	(*****P14_BadBottleConyevor********)
	bBadBottleConveyorEnable						:BOOL;									//Zezwolenie na pracę transportera odrzuconych butelek
	nBadBottleConveyorVelocitySV					:UINT;									// Predkosc zadana transportera
	bBadBottleConveyorStart							:BOOL; 									// Zezwolenie na pracę transportera we/wy	

	(*******P14_TurnTable********)
	bExitTurnTableEnable							:BOOL;(**)								//Zezwolenie na pracę etykieciarki
	bExitTurnTableCmdStart 							:BOOL;
	bExitTurnTableGateRun							:BOOL;
	bExitConveyorEnable								:BOOL;(**)								//Zezwolenie na pracę 
	nExitConveyorVelocitySV							:UINT;
	bExitConveyorCmdStart 							:BOOL;
	bExitConveyorGateRun							:BOOL;

	
	(********P15_FormTransporters********)
	bFormTransportersEnable							:BOOL;			
	bFormTransportersDispencerCmdStart				:BOOL; 									// Start transporterów formatek w cyklu
	bFormTransportersBeforeROPPCmdStart				:BOOL;
	bFormTransportersScrewerCmdStart				:BOOL; 									// Start transporterów formatek w cyklu
	bFormTransportersScrewerStop					:BOOL; 									// Start transporterów formatek w cyklu
	bFormTransportersBeforeROPPStop					:BOOL;
	bFormTransportersDispencerSlowSpeedPulse		:BOOL;									// Wolna prędkość transportera
	bFormTransportersDispencerSlowSpeed				:BOOL;									// Wolna prędkość transportera
	bFormTransportersDispencerResetSpeed			:BOOL;									// Reset prędkości transportra
	ulFormTransportersScrewerSlowNumber				:ULINT;									// Nr RFID ostatniej formatki bez korka
	bFormTransportersAfterCapSorterCmdStart			:BOOL;									// Start transportera przez zakręcarka								// Aktywacja
	bFormTransportersBeforeScrewerCmdStart			:BOOL;									// Start transportera przez zakręcarka								// Aktywacja
	bFormTransporterSlowerCmdStart					:BOOL;									// Start transportera spowalniacza fomatek
	bFormTransportersAfterScrewerCmdStart			:BOOL;									// Start transportera przez zakręcarka								// Aktywacja
	ulSingleRealeseIfNoCapFromScrewersNumber		:ULINT;									// Nr RFID ostatniej formatki bez korka
	bSingleRealeseIfNoCapFromScrewersPulse			:BOOL;
	iSingleRealeseIfNoCapFromScrewersPulse			:INT;
				
	//Opcja z falownikiem
	nFormTransportersDispencerVelocitySV			:UDINT;		// Prędkość transportera otwartych butelek
	nFormTransportersScrewerVelocitySV				:UDINT;		// Prędkość transportera zamkniętych butelek
	nFormTransportersAfterCapSorterVelocitySV		:UDINT;		// Prędkość transportera przed zakręcarkami
	nFormTransportersBeforeScrewerVelocitySV		:UDINT;		// Prędkość transportera przed zakręcarkami
	nFormTransportersSlowerVelocitySV				:UDINT;		// Prędkość spowalniacza
	nFormTransportersAfterScrewerVelocitySV			:UDINT;		// Prędkość transportera przed zakręcarkami
	nFormTransportersROPPVelocitySV					:UDINT;		// Prędkość spowalniacza

	(******P16_LabelMachine********)
	bLabelMachineEnable								:BOOL;(**)								//Zezwolenie na pracę etykieciarki
	bLabelMachineCmdStart							:BOOL;		

	(*****P17_CircularInkJet********)
	bCircularInkjetEnable 							:BOOL;									// Zezwolenie na pracę Inkjet'u obwodowego	
	iCircularInkjetSpeed 							:INT;									// Prędkość rolek
	iCircularInkjetDelay							:INT;									// Opóźnienie docisku rolek
	iCircularInkjetHold								:INT;		
	
	bDragingFormsNotDone							:BOOL;				//Zmienna pomocnicza od przeciagania

	(**P20_ExhaustFan**)
	bExhaustFanEnable								:BOOL;
	bExhaustFanCmdStart								:BOOL;
	udiExhaustFanVelocitySV							:UDINT;
	


END_VAR

VAR_GLOBAL PERSISTENT
	(*****Zmienne presistent****)
	
	(***MAIN***)
	eRFID											:ARRAY [1..100] OF S_PackageState;		// STRUKTURA RFID
	AbRFIDFormOrder									:ARRAY [0..100] OF ULINT;				// Globalny rejestr kolejności formatek

	// Auton
	iDispencerRepair1								:INT;
	itonAfterDispencersRepair						:INT;
	itonAfterDispencersRepair1B						:INT;
	itonAfterDispencersRepair2						:INT;	
	itonAfterDispencersRepair3						:INT;	
	itonAfterDispencersRepair4						:INT;	
	itonRobotBottleTransferedToLabelerRepair		:INT;
	itonRobotBottleTransferedToLabeler2Repair		:INT;
	
	(***P00_Counters***)
	nGlobalCounterTemp								:UDINT;									//Tymczasowa zmienna do zapisywania licznika globalnego do pliku raz na jakiś czas
	
	(*Do diagnostyki*)
	iCounterDispencer34DosingAborted				:INT;
	iRepairFormBeforeDispenscerCounter				:INT;
	iRepairFormBeforeDispenscer2PhaseCounter		:INT;
	iRepairAfterDispencerCounter					:INT;
	iRepairBeforeDispencer12Counter					:INT;
	iRepairBeforeDispencer12Counter2				:INT;	
	iWeightRepair1Counter							:INT;
	iWeightRepair2Counter							:INT;
	iRepairFourthFormBeforeDispencerCounter			:INT;
	iRepairBeforeDispencer34Counter					:INT;
	
	iRepairLidFeeder1Counter						:INT;
	iRepairLidFeeder2Counter						:INT;
	iRepairLidFeeder3Counter						:INT;
	iRepairLidFeeder4Counter						:INT;
	
	iUnderScrewerPackageState222nCardNumberChangeCounter		: INT;
	iUnderScrewerPackageState333nCardNumberChangeCounter		: INT;
	iUnderScrewerPackageState111nCardNumberChangeCounter		: INT;
	
	iDispencerPackageState4nCardNumberChangeCounter	:INT;		
	iDispencerPackageState3nCardNumberChangeCounter	:INT;	
	iDispencerPackageState2nCardNumberChangeCounter	:INT;	
	iDispencerPackageState1nCardNumberChangeCounter	:INT;	
	
	iRobotPackageState2nCardNumberChangeCounter		:INT;	
	iRobotPackageState1nCardNumberChangeCounter		:INT;	
	
	iRobotRepairPackageForm1Counter					:INT;
	iRobotRepairPackageForm2Counter					:INT;	
	
	iScrewerFormStuck								:INT;
	iScrewerFormStuck2								:INT;
	iScrewerFormStuck3								:INT;

	(***MAIN***)
	//aSetIDBottle
	nID												:UDINT;									// Identycikacja butelek
		
	(*****P02_Dispencers****)
	bTank1LevelSensorCalibrated						:BOOL;									//Czujnik poziomu nr 1 skalibrowany	
	
	(*****P13_BottleTransfer********)
	nBottleTransferLubricationCounter				:DINT;									//Licznik po którym wyświetla się ostrzeżenie o smarowaniu robota
	
	
END_VAR

// ---- GVLs/gvlChecks.TcGVL
(*
Nazwa:			GVL_Checks
Opis:			Zmienne do sprawdzania błędów
Wersja:			v0.1
Data:			2018-10-10
Autor:			DP
Urzadzenia:		
Konfiguracja:	
Info:
(*d*) - obslużone
*)

{attribute 'qualified_only'}
VAR_GLOBAL PERSISTENT
	dCheckBounds		: DINT;	(*Licznik przekroczen zakresu indexow, np. tablic*)
	dCheckDivDInt		: DINT;	(*Licznik prob dzielenia Dint przez 0*)
	dCheckDivLInt		: DINT; (*Licznik prob dzielenia LInt przez 0*)
	dCheckDivLReal		: DINT; (*Licznik prob dzielenia LREAL przez 0*)
	dCheckDivReal		: DINT; (*Licznik prob dzielenia REAL przez 0*)
	dCheckRangeSigned	: DINT;	(*Licznik przekroczen  liczby znakowej*)
	dCheckRangeUnsigned	: DINT; (*Licznik przekroczen  liczby bezznakowej*)
END_VAR

// ---- GVLs/gvlCommunication.TcGVL
VAR_GLOBAL
	
		(*****P01_BottleSorter********)	
		stBottleSorterWrite			AT %MB0		: ST_Communication;		//Wysyłane zmienne do BottleSorter	
		//stBottleSorterWrite		AT %Q*		: ST_Communication;		//Wysyłane zmienne do BottleSorter
		stBottleSorterRead			AT %I*		: ST_Communication;		//Odczytane zmienne z BottleSorter
		
		//Zapis ADS
		//nic nie potrzeba, sprawdzanie czy jest butelka 
		//jest przed dozownikami
		
		//Odczyt ADS
		//nic nie potrzeba, sprawdzanie czy jest butelka 
		//jest przed dozownikami	
		bBottleSorterDoor1Open						: BOOL;				// Drzwi 1 otwarte
		bBottleSorterDoor2Open						: BOOL;				// Drzwi 2 otwarte	
		bBottleSorterSystemDiagError				: BOOL;				// Bład systemu BottleSorter

		(*****P04_CapSorter********)	
		stCapSorterWrite			AT %MB2000	: ST_Communication;	//Wysyłane zmienne do CapSorter	
		//stCapSorterWrite			AT %Q*		: ST_Communication;		//Wysyłane zmienne do CapSorter	
		stCapSorterRead				AT %I*		: ST_Communication;		//Odczytane zmienne z CapSorter
		
		//Zapis ADS		
		bCapSorterRobotPlace					: BOOL;				// Nałóż nasadki	
		bCapSorterRobotBottleAndNoCap1			: BOOL;				// Jest butelka bez nasadki w formatce 1
		bCapSorterRobotBottleAndNoCap2			: BOOL;				// Jest butelka bez nasadki	w formatce 2
		bCapSorterRobotBottleAndNoCap3			: BOOL;				// Jest butelka bez nasadki w formatce 3
		bCapSorterRobotBottleAndNoCap4			: BOOL;				// Jest butelka bez nasadki w formatce 4
		bCapSorterRobotPreparePlace				: BOOL;				// Przygotuj nasadki 			
		bCapSorterBeforeRobotBottleAndNoCap1	: BOOL;				// Jest butelka bez nasadki w formatce 1 przed robotem
		bCapSorterBeforeRobotBottleAndNoCap2	: BOOL;				// Jest butelka bez nasadki	w formatce 2 przed robotem
		bCapSorterBeforeRobotBottleAndNoCap3	: BOOL;				// Jest butelka bez nasadki w formatce 3 przed robotem
		bCapSorterBeforeRobotBottleAndNoCap4	: BOOL;				// Jest butelka bez nasadki w formatce 4 przed robotem
		
		//Odczyt ADS
		bCapSorterRobotPlaceDone				: BOOL;				// Wykonano, formatki mogą odjechać			
		bCapSorterRobotForm1CapPutted			: BOOL;				// Nasadka nałożona
		bCapSorterRobotForm2CapPutted			: BOOL;				// Nasadka nałożona
		bCapSorterRobotForm3CapPutted			: BOOL;				// Nasadka nałożona
		bCapSorterRobotForm4CapPutted			: BOOL;				// Nasadka nałożona
		
		bCapSorterDoor1Open						: BOOL;				// Drzwi 1 otwarte
		bCapSorterDoor2Open						: BOOL;				// Drzwi 2 otwarte		
		bCapSorterDoor3Open						: BOOL;				// Drzwi 3 otwarte	
		bCapSorterDoor4Open						: BOOL;				// Drzwi 4 otwarte		
		
		bCapSorterEmergencyStopButton1Pressed	: BOOL;				// Drzwi 1 otwarte
		bCapSorterEmergencyStopButton2Pressed	: BOOL;				// Drzwi 2 otwarte		
		bCapSorterEmergencyStopButton3Pressed	: BOOL;				// Drzwi 3 otwarte	
		
		bCapSorterRobotPlaceAck					: BOOL;				// Potwierdzenie rozpoczęcia cyklu		
	
END_VAR

// ---- GVLs/GVL_CP.TcGVL

VAR_GLOBAL
	

	//MAIN/PACKML
	eCapPusherPackageState					:ARRAY [1..17] OF S_PackageState;		// [1..6] 

	(******P00_Alarms******)
	CapPusherGateError						:S_Error; 								// Szlaban
	CapPusherFeederError					:S_Error; 								// Podajnik
	CapPusherError							:S_Error;								// Wbijak

	(******P07_CapPusher********)	  

	//Szlaban
	bCapPusherGateRun						:BOOL;		

	//Podajnik
	bCapPusherFeederDoHoming				:BOOL;									// Wykonanie bazowania stacji podajnika 
	iCapPusherFeederTimeDelayOn				:INT; 										
	iCapPusherFeederTimeDelayOff			:INT; 
	iCapPusherFeederTimeToEmptySleeveError	:INT:=120;									// Czas do alarmu pustego rękawa 
	iCapPusherFeederCheckCountNOK			:INT;									// Zliczanie butelek bez nasadek

	//Zakrecanie
	bCapPusherDoHoming						:BOOL;									// Wykonanie bazowania stacji 
	bCapPusherEnable						:BOOL:=TRUE; 	
	iCapPusherTime							:INT; 	
	iCapPusherTime2							:INT;	

END_VAR

(*
VAR_GLOBAL PERSISTENT
	iRepairROPP1Counter						:INT;
	iRepairROPP2Counter						:INT;
	iRepairROPP3Counter						:INT;
	iRepairROPP4Counter						:INT;
END_VAR	*)

// ---- GVLs/GVL_IO.TcGVL
(*
Nazwa:			GVL_IO
Opis:			Zmienne I/O nie wykorzystywane w blokach stacji
Wersja:			v0.1
Data:			2018-10-10
Autor:			DP
Urzadzenia:		
Konfiguracja:	
Info:
(*d*) - obslużone
*)


VAR_GLOBAL

(*Safety ##############################*)
	//Przesylane, odbierane z/do SafetyPLC
	IbEmergencyStopButton 	AT %I*		: BOOL; 		//Jeśli FALSE - Estop wysyołany przez przyciski
	IbEmergencyStop 		AT %I* 		: BOOL; 		//Jeśli TRUE - maszyna w stanie bezpiecznym, FALSE - EStop
	IbBottleFeederSafety	AT %I*		: BOOL;			// Status Safety z podajnika butelek
	IbSafetyResetIn			AT %I*		: BOOL;			// Przycisk Reset
	QbSafetyResetCapSorterIn AT %Q*		: BOOL;			// Przycisk Reset
	QbSafetyResetBottleSorterIn AT %Q*	: BOOL;			// Przycisk Reset
	QbSafetyResetDelay 		AT %Q*		: BOOL;			// Zezwolenie na pierwsze zresetowanie
	
	
	IbCommunicationErrorUF50	AT %I* 	:BOOL;			//Do alarmu komunikacji z safety
	IbCommunicationErrorUP50B	AT %I* 	:BOOL;			//Do alarmu komunikacji z safety
	
	IbBottleSorterDisable		AT %I* 	:BOOL:=TRUE;			//Sygnał z kluczyka blokady safety
	IbCapSorterDisable			AT %I* 	:BOOL:=TRUE;			//Sygnał z kluczyka blokady safety

	
(*Wejscia ogólne #####################*)

	IbPowerSupplyOK 				AT %I*		:BOOL;		//Napięcie zasilania OK
	IbDCSupply1OK 					AT %I*		:BOOL;		//Zasilacz alarm	
	IbFuseFB1OK						AT %I*		:BOOL;		//Bezpiecznik FB1 przepalony
	IbDCSupply2OK					AT %I*		:BOOL;		//Zasilacz alarm	
	IbFuseFB2OK						AT %I*		:BOOL;		//Bezpiecznik FB2 przepalony
	IbDCSupply3OK					AT %I*		:BOOL;		//Zasilacz alarm	
	IbFuseDrivesOK					AT %I*		:BOOL;		//Bezpiecznik Servonapędów
	IbFuseFormTransporter1OK		AT %I*		:BOOL;		//Bezpiecznik silnikowe napędu transportera 1
	IbFuseFormTransporter2OK		AT %I*		:BOOL;		//Bezpiecznik silnikowe napędu transportera 2
	IbFuseFormTransporter3OK		AT %I*		:BOOL;		//Bezpiecznik silnikowe napędu transportera 3 (odrzuty)
	IbFuseFormTransporter4OK		AT %I*		:BOOL;		//Bezpiecznik silnikowe napędu transportera 4 (spowalniacz)
	IbFuseFormTransporter5OK		AT %I*		:BOOL;		//Bezpiecznik silnikowe napędu transportera 4 (33F1)
	IbFuseFormTransporter6OK		AT %I*		:BOOL;		//Bezpiecznik silnikowe napędu transportera 4 (34F1)
	IbBottleFeederTurntableOK		AT %I*		:BOOL;		//Zabezpieczenie silnikowe stolu obrtooergo
	IbDCSupply4OK					AT %I*		:BOOL;		//Zasilacz alarm			
	IbDCSupply5OK					AT %I*		:BOOL;		//Zasilacz alarm		
	IbFuseFB3OK						AT %I*		:BOOL;		//Bezpiecznik FB3 przepalony
	IbDC5VSupply1OK 				AT %I*		:BOOL;		//Zasilacz 5V alarm	

	
	IbLinearPowerSupplyOK			AT %I*		:BOOL;	
	IbStepperPowerSupplyOK			AT %I*		:BOOL;	
	IbFuseFanEXMotor				AT %I*		:BOOL;	
	IbStepperMotorsFuseOK			AT %I*		:BOOL;
	IbFuse10F9OK					AT %I*		:BOOL;
	IbFuse10F11OK					AT %I*		:BOOL;
	
	//IbFuseTankMixerEngineOK w Dispencers
	IbTanksDoorsOpen 				AT %I*		:BOOL;		//Otwarte drzwi pod zbiornikami
	IbLidSealingDoorsOpen			AT %I*		:BOOL;		//Otwarte drzwi przygrzewaczki
	IbGripperScrewerDoorsOpen		AT %I*		:BOOL;		//Otwarte drzwi przy zakrecarkach
	IbDispencersDoorsOpen 			AT %I*		:BOOL;		//Otwarte drzwi przy dozownikach
	IbBottleTransferDoorsOpen		AT %I*		:BOOL;		//Otwarte drzwi z boku dozowników

	IbEmergencyStopButton0Pressed	AT %I*		:BOOL;		//Przyciśnięty przycisk E-Stop0	Pulpit główny przod
	IbEmergencyStopButton1Pressed	AT %I*		:BOOL;		//Przyciśnięty przycisk E-Stop1 przy transporterze odrzuconych opakowań
	IbEmergencyStopButton2Pressed	AT %I*		:BOOL;		//Przyciśnięty przycisk E-Stop2 przy drzwiach robota
	IbEmergencyStopButton3Pressed	AT %I*		:BOOL;		//Przyciśnięty przycisk E-Stop3 przy zakręcarkach
	IbEmergencyStopButton4Pressed	AT %I*		:BOOL;		//Przyciśnięty przycisk E-Stop4	Pulpit tylny

	// podajnik butelek
	
	IbBottleFeederSafetyDoor1Open	AT %I*		:BOOL;		// Czujnik otwarcia drzwi dostępowych 
	IbBottleFeederSafetyDoor2Open	AT %I*		:BOOL;		// Czujnik otwarcia drzwi dostępowych drugie
	IbBottleFeederSafetyDoor3Open	AT %I*		:BOOL;		// Czujnik otwarcia drzwi dostępowych drugie
	
	
	//Vasyl 28.05
	IbPucksInserterRollerFuse		 AT %I*      :BOOL;		// Zabezpieczenie 71F4 Rolka obracająca
	IbPucksInserterPushTableFuse	 AT %I*      :BOOL;		// Zabezpieczenie 71F3 Stół podający
	IbEmergencyStopButtonPushtable1  AT %I*		:BOOL;
	IbEmergencyStopButtonPushtable2  AT %I*		:BOOL;
	
	
	IbCycleStartButton				AT %I*		:BOOL;		//Przycisk Startu cyklu
	//IbSafetyResetIn				AT %I*		:BOOL;		//Reset
	IbCycleStopButton				AT %I*		:BOOL;		//Przycisk Stopu cyklu
	//IbTank1LevelLow w Dispencers
	//IbTank2LevelLow w Dispencers
	IbCompressedAirOK 				AT %I*		:BOOL;		//Zasilanie powietrzem sprężonym OK	
	
(* I/O robot*)
	//Alarm zasilacz DC1 w BottleTransfer
	//Bezpiecznieki OK w BottleTransfer

	IbFuseCircularInkjetOK			AT %I*		:BOOL;		//Zabezpieczenie silnikowe InkJet obwodowy	
	
	QbResetFuseFB1					AT %Q*		:BOOL;	
	QbResetFuseFB2					AT %Q*		:BOOL;
	QbResetFuseFB3					AT %Q*		:BOOL;	

(* Diagnostyka modułów*)
	IbPowerSuppyTerminal1UpUndervoltage	AT %I*		:BOOL;	{warning 'dodać alarm'}// Brak napięcia zasilania na module ST1 w szafie głównej
	IbPowerSuppyTerminal1UsUndervoltage	AT %I*		:BOOL;	
	IbPowerSuppyTerminal2UpUndervoltage	AT %I*		:BOOL;	// Brak napięcia zasilania na module ST1 w szafie robota
	IbPowerSuppyTerminal2UsUndervoltage	AT %I*		:BOOL;	// Brak napięcia E-Bus na module ST1 w szafie robota
	
	QbDispencersDoorsClose				AT %Q*		:BOOL;		// Rozkaz zamkniecia 
	QbGripperScrewerClose				AT %Q* 		:BOOL;		// Rozkaz zamkniecia 
	QbBottleTransferDoorsClose			AT %Q*		:BOOL; 		// Rozkaz zamkniecia 
	QbTanksDoorsClose 					AT %Q*		:BOOL;		// Rozkaz zamkniecia
	QbLidSealingDoorsClose				AT %Q*		:BOOL;		// Rozkaz zamkniecia
	
	(*Wybdmuch nakretek*)
	QbBlowAfterGripperScrewer						: BOOL; 
	QbBlowBeforeGripperScrewer						: BOOL; 
	IbBlowBeforeGripperScrewerSensor				: BOOL;
	QbGateBeforeGripperScrewer						: BOOL;	
	IbGateBeforeGripperScrewerSensor				AT %I*		:BOOL;	

	//Dodatkowy szlaban przed zakrecarka
	QbGripperScrewerStoperActuator			:BOOL;	//Stoper
	QbGripperScrewerStoper2Actuator			:BOOL;	//Stoper krótki
	QbGripperScrewerGateBeforeActuator		:BOOL;	//Szlaban
	//Koniec Dodatkowy szlaban przed zakrecarka

	//Dodatkowy szlaban za robotem
	QbBottleTransferAfterDragActuator		:BOOL;	//Stoper
	QbBottleTransferAfterDragStoperActuator	:BOOL;	//Stoper krótki
	QbBottleTransferAfterDragGateActuator	:BOOL;	//Szlaban
	//Koniec Dodatkowy szlaban za robotem


	
	//Dodatkowy popychacz za zakręcarką
	QbGripperScrewerAcceleratorActuator			:BOOL;
	
	(*I/O TurnTable*)
	IbTurnTableSafety						AT %I*		:BOOL;		//Przyciśnięty przycisk E-Stop0	Pulpit główny
	IbTurnTableMotorOK						AT %I*		:BOOL;		//Zabezpieczenie silnikowe stolu obrtooergo 
	IbTurnTableEmergencyStopButtonPressed	AT %I*		:BOOL;		//Przyciśnięty przycisk E-Stop0	Pulpit główny
	IbTurnTableCycleStartButton				AT %I*		:BOOL;		//Przycisk Startu cyklu
	IbTurnTableCycleStopButton				AT %I*		:BOOL;		//Przycisk Stopu cyklu
	IbTurnTableFuseProtection				AT %I*		:BOOL;		//Zabezpieczenie stół obrotowy

	IbExitConveyorOK						AT %I*		:BOOL;		//Zabezpieczenie silnikowe stolu obrtooergo


	(*I/O PI*)
	IbPucksInserterDoorsOpen	{warning 'PI'}	AT %I*		:BOOL;		//Otwarte drzwi podajnika opakowań
	QbPickInserterDoorsClose	{warning 'PI'}	AT %Q*		:BOOL;		// Rozkaz zamkniecia 
	IbPucksInserterEmergencyStopButton0Pressed	AT %I*		:BOOL;		//Przyciśnięty przycisk E-Stop0	
	IbPucksInserterEmergencyStopButton1Pressed	AT %I*		:BOOL;		//Przyciśnięty przycisk E-Stop1	
	IbPucksInserterCycleStartButton				AT %I*		:BOOL;		//Przycisk Startu cyklu
	IbPucksInserterCycleStopButton				AT %I*		:BOOL;		//Przycisk Stopu cyklu

(* IO wybychowe**)
	
	IbExModeSwitchNormalMode		AT %I*		:BOOL;		// Wybór trybu pracy - tryb zwykły
	IbExModeSwitchExMode			AT %I*		: BOOL;		// Wybór trybu pracy - tryb pracy wybuchowej
	
	
(* Czujnik ciśnienia w układzie *)
	IbPressureInSystemSensor		AT %I*	:BOOL;
	

END_VAR

// ---- GVLs/GVL_ROPP.TcGVL

VAR_GLOBAL
	

	//MAIN/PACKML
	eBeforeROPPCapControlPackageState		:ARRAY [1..17] OF S_PackageState;		// [1..1] 
	eBeforeROPPPackageState					:ARRAY [1..17] OF S_PackageState;		// [1..6] 
	eBeforeROPP2PackageState				:ARRAY [1..17] OF S_PackageState;		// [1..6] 
	eUnderROPPPackageState 					:ARRAY [1..17] OF S_PackageState;		// [1..3] 
	eUnderROPPCorrectCapPackageState		:ARRAY [1..17] OF S_PackageState;		// [1..7] 

	(******P00_Alarms******)
	ROPPSlowerError							:S_Error; 								// Spowalniacz
	ROPPFeederError							:S_Error; 								// Spowalniacz
	ROPPDragError							:S_Error;								// 14 
	ROPPCappingError						:S_Error;								// 14 

	(******P07_ROPP********)	  

	//Spowalniacz
	bROPPSlowerEnable						:BOOL:=TRUE;			
	bROPPSlowerCmdStart						:BOOL:=TRUE;									// Start transportera spowalniacza fomatek
	nROPPSlowerVelocitySV					:UDINT:=2100;	

	//Podajnik
	bROPPFeederDoHoming						:BOOL;									// Wykonanie bazowania stacji podajnika 
	bROPPFeederEnable						:BOOL; 	
    lrROPPFeederHeightPosSV					:LREAL;									 	
	iROPPFeederTimeDelayOn					:INT; 										
	iROPPFeederTimeDelayOff					:INT; 
	iROPPFeederTimeToEmptySleeveError		:INT;									// Czas do alarmu pustego rękawa 
	iROPPFeederCheckCountNOK				:INT;									// Zliczanie butelek bez nasadek

	//Przeciąganie formatek 
	aROPPDragAxisRef						:AXIS_REF;								// Struktura osi napędu krokowego przeciągania	
	bROPPDragEnable							:BOOL;									// Zezwolenie na pracę przeciągania 
	bROPPDragDoHoming						:BOOL;									// Wykonanie bazowania przeciągania
	bROPPDragHeightSet						:BOOL;									// Wykonanie bazowania przeciągania
	bROPPDragPrepareRun						:BOOL;
	lrROPPDragVelocity						:LREAL:=100;							// Prędkośc przeciągania
	lrROPPDragAcceleration					:LREAL:=12;								// Przyspieszenie przeciągania
	lrROPPDragDeceleration					:LREAL:=15;								// Hamowanie przeciągania

	//Zakrecanie
	bROPPCappingRunEngine					:BOOL;									
	bROPPCappingDoHoming					:BOOL;									// Wykonanie bazowania stacji 
	bROPPCappingEnable						:BOOL; 	
    lrROPPCappingHeightPosSV				:LREAL;									 	
	lrROPPCappingVelocitySV					:UDINT;	
	iROPPCappingTime						:INT; 	
	iROPPCappingTime2						:INT;	
	iROPPCapping1Tool						:INT;									// Wybór narzędzia (1-5), opisy w tablicy AsGripperScrewerTool	

END_VAR

(*
VAR_GLOBAL PERSISTENT
	iRepairROPP1Counter						:INT;
	iRepairROPP2Counter						:INT;
	iRepairROPP3Counter						:INT;
	iRepairROPP4Counter						:INT;
END_VAR	*)

// ---- GVLs/GVL_RS.TcGVL

VAR_GLOBAL
	
	//MAIN/PACKML
	eRollerScrewerPackageState					:ARRAY [1..17] OF S_PackageState;		// [1..6] 

	(******P00_Alarms******)
	RollerScrewerGateError						:S_Error; 								
	RollerScrewerError							:S_Error;								
	RollerScrewerCatchError						:S_Error;								
                                                                                        
	(*****P11_RollerScrewer********)  
	//Szlaban
	bRollerScrewerGateRun						:BOOL;		
	//Zakrecanie
	bRollerScrewerDoHoming						:BOOL;									// Wykonanie bazowania stacji podajnika 
	//Ciśnienia - nie wiadomo czy będą
	lrRollerScrewerCatchPressure 				:LREAL;			
	lrRollerScrewerPressingRollsPressure		:LREAL;			
	lrRollerScrewerPressingTopPressure 			:LREAL;			
	//Zakręcarka rolkowa
	aRollerScrewerFrontAxisRef					: AXIS_REF;									// Struktura NC napędu zakręcarki rolkowej
	aRollerScrewerRearAxisRef					: AXIS_REF;									// Struktura NC napędu zakręcarki rolkowej
	bRollerScrewerEnable						: BOOL;			
	bRollerScrewerFindScrew						: BOOL; 		
	lrRollerScrewerFindingScrewDegree			: LREAL; 		
	lrRollerScrewerVelocity						: LREAL:=50; 
	iRollerScrewerTightTime						: INT:=100;  
	lrRollerScrewingTightTorque					: LREAL;  		
    lrRollerScrewerHeightPosSV					: LREAL:=72;	
	uiRollerScrewerTopActuatorTimeDelayOff		: UINT;  		
	//Chwytak zakręcarki rolkowej                               		
	lrRollerScrewerCatchHeightSV				: LREAL:=36; 
	bRollerScrewerCatchRun						: BOOL; 
	bRollerScrewerCatchDoHoming					: BOOL; 

	
END_VAR

(*
VAR_GLOBAL PERSISTENT
	iRepairROPP1Counter						:INT;
	iRepairROPP2Counter						:INT;
	iRepairROPP3Counter						:INT;
	iRepairROPP4Counter						:INT;
END_VAR	*)

// ---- GVLs/Iterators.TcGVL
VAR_GLOBAL
	i								: INT;
END_VAR

// ---- GVLs/UVFF/GVL_Recipe.TcGVL
(*
Nazwa:			GVL_Recipe
Opis:			Zmienne recepturowe tylko do wizualizacji
Wersja:			v0.2
Data:			2024-02-20
Autor:			MK
Urzadzenia:		
Konfiguracja:	
Info:
Zmiany:
- 20240220 [DP] Poprawki przed nowa wizką
*)
VAR_GLOBAL
	(*Legenda dla wizki :
		[H] - Hidden, prawdopodobnie nie potrzebne
		[I] - Info, informacja,
		[L] - Later, do zrobienia później, być może do przerobienia
		Uprawienia:
		brak opisu - operator
		[m] - Meechanik i powyżej
		[t] - Technolog i powyżej
		[s] - Serwis i powyżek
		[a] - Admin			
	*)	
	
	//Sorter nasadek, typ produktu	
	iCapSorterProductType										: INT		:= 2; 		//		Typ produktu: 0- kule/fliptopy, 1- pompki, 2- disctop, 3-airless, 4-decoration cap (wyłączone podcisnienie na załapywarce), 5- decoration cap with new gripper (wyłączone podcisnienie + nowy program do robota)
	uiCapSorterIndexShow										: UDINT		:= 5;		//		Index produktu	
	bPresenceBottleEnableShow									: BOOL;					//		Sprawdzanie butelki w formatce

//--------------------------------------CapSorterTransporter-----------------------------------------------------------------------------------------------------------------------------	
	// Sorter nasadek, transporter zasobnika
	bCapSorterTransporterEnableShow								: BOOL;					//		Aktywacja
	iCapSorterTransporterTankConveyorVelocityShow				: INT		:= 1200;	//		Prędkość 							| [%] (1.0-100.0)
	iCapSorterTransporterStartDelayTimeShow						: INT		:= 100;		//		Timer do załączania 				| [ms] (0.0-10_000.0)
	udiCapSorterTransporterTimeProductOnSensorBeforeBrushShow	: UDINT		:= 150;		//		Timer pracy							| [ms] (0.0-10_000.0)
	iCapSorterTransporterEmptyingConveyorSpeedShow				: INT		:= 25;		// 		Prędkość, opróżnianie 				| [%] (1.0-100.0)
	iCapSorterTransporterVolumeOfCapsShow						: INT		:= 330;		//		Odłegłość do zamknięć, ostrzeżenie 	| [mm] (0.0-10_000.0)

//---------------------------------------CapSorterWheel----------------------------------------------------------------------------------------------------------------------------	
	// Sorter nasadek, stól
	bCapSorterWheelEnableShow									: BOOL;					//		Aktywacja
	lrCapSorterWheelMoveAccelerationEmptyTableShow				: LREAL		:= 5000;	//		Dynamika rozpędzania - pusty 		| [obr/min²], (1.0-100_000.0) 
	lrCapSorterWheelMoveDecelerationEmptyTableShow				: LREAL		:= 5000;    //		Dynamika spowalniania - pusty 		| [obr/min²] (1.0-100_000.0) 
	lrCapSorterWheelMoveSpeedEmptyTableShow						: LREAL		:= 334;     //		Prędkość - pusty 					| [obr/min] (1.0-10_000.0)                
	lrCapSorterWheelMoveAngleEmptyTableShow						: LREAL		:= 20;      //		Kąt - pusty 						| [obr/min] (0.0-360.0)                        
	lrCapSorterWheelJerkAngleEmptyTableShow						: LREAL		:= 15000;   //		Zryw - pusty 						| [obr/min³] (1.0-1_000_000)                  
	iCapSorterWheelWaitingAfterRotationEmptyTableShow			: INT		:= 100;     //		Czas stabilizacji - pusty 			| [ms] (0.0-1_000)                 
	
	lrCapSorterWheelMoveAccelerationFullTableShow				: LREAL		:= 5000;	//		Dynamika rozpędzania - pełny 		| [obr/min²], (1.0-100_000.0) 
	lrCapSorterWheelMoveDecelerationFullTableShow				: LREAL		:= 5000;    //		Dynamika spowalniania - pełny 		| [obr/min²] (1.0-100_000.0) 
	lrCapSorterWheelMoveSpeedFullTableShow						: LREAL		:= 334;     //		Prędkość - pełny 					| [obr/min] (1.0-10_000.0)                
	lrCapSorterWheelMoveAngleFullyTableShow						: LREAL		:= 6;       //		Kąt - pełny 						| [obr/min] (0.0-360.0)                        
	lrCapSorterWheelJerkAngleFullTableShow						: LREAL		:= 15000;   //		Zryw - pełny 						| [obr/min³] (1.0-1_000_000)                  
	iCapSorterWheelWaitingAfterRotationFullTableShow			: INT		:= 30;      //		Czas stabilizacji - pełny 			| [ms] (0.0-1_000)                 
	
	lrCapSorterWheelMoveAccelerationHalfFullTableShow			: LREAL		:= 5000;	//		Dynamika rozpędzania - półpełny 	| [obr/min²], (1.0-100_000.0) 
	lrCapSorterWheelMoveDecelerationHalfFullTableShow			: LREAL		:= 5000;    //		Dynamika spowalniania - półpełny 	| [obr/min²] (1.0-100_000.0) 
	lrCapSorterWheelMoveSpeedHalfFullTableShow					: LREAL		:= 334;     //		Prędkość - półpełny 				| [obr/min] (1.0-10_000.0)                
	lrCapSorterWheelMoveAngleHalfFullyTableShow					: LREAL		:= 12;      //		Kąt - półpełny						| [obr/min] (0.0-360.0)                        
	lrCapSorterWheelJerkAngleHalfFullTableShow					: LREAL		:= 15000;   //		Zryw - półpełny 					| [obr/min³] (1.0-1_000_000)                  
	iCapSorterWheelWaitingAfterRotationHalfFullTableShow		: INT		:= 50;      //		Czas stabilizacji - półpełny 		| [ms] (0.0-1_000)               
	
//-------------------------------------CapSorterCamera------------------------------------------------------------------------------------------------------------------------------	                                                    	
	// Sorter nasadek, system wizyjny
	
    bCapSorterCameraEnableShow									: BOOL; 				//	[H]	Aktywacja                            	
	
//-----------------------------------------CapSorterRobot--------------------------------------------------------------------------------------------------------------------------	
	// Sorter nasadek, robot
	bCapSorterRobotEnableShow									: BOOL;					//		Aktywacja
                                                                                                                           	
	lrCapSorterRobotPlace1PositionXShow							: LREAL;				//		Offset odkładania 1, X 			| [mm]	((-100.0)-100.0)       
	lrCapSorterRobotPlace1PositionYShow							: lreal;    			//		Offset odkładania 1, Y 			| [mm]	((-100.0)-100.0)       
	lrCapSorterRobotPlace1PositionZShow							: lreal;    			//		Offset odkładania 1, Z 			| [mm]	((-100.0)-100.0)       
	lrCapSorterRobotPlace1PositionCShow							: lreal;    			//		Offset odkładania 1, C 			| [° ]	((-360.0)-360.0)                 
	iCapSorterRobotPickElevationShow							: INT;					//		Punkt nad poz. Pick				| [mm]	(30-1000)
	iCapSorterRobotPickTimeShow									: INT;					//		Czas przyssania					| [ms]	(0-10_000)
	iCapSorterRobotVacuumActivationShow							: INT;					//		Czas przed przyssaniem			| [ms]	(0-1000)
	iCapSorterRobotVacuumOffShow								: INT;					//		Czas przed oddmuchem			| [ms]	(0-1000)
	iCapSorterRobotPlaceTimeShow								: INT;					//		Czas oddmuchu					| [ms]	(0-1000)
	iCapSorterRobotTCP_PlaceOffsetShow							: INT;					//		Wysokość od TCP do p. odłożenia	| [mm]	(0-1000)									
	iCapSorterRobotAccelerationDecelerationShow					: INT;					//		Dynamika rozpędzania/hamowania	| [%]	(20-100)
	iCapSorterRobotGripperWatchdogShow							: INT;					//		Czas sprawdzania silownika		| [ms]	(0-1000)
	iCapSorterRobotParalaxCorrectionShow						: INT;					//		Korekta paralaxy				| [mm]	(0-100)
	
	iCapSorterRobotNumberToolShow								: INT;					//		Numer narzędzia					| 		(0-10)
	iCapSorterRobotPickPositionZShow							: INT;					//		Wysokość pobierania 			| [mm]	(0-200)
	iCapSorterRobotTCP_Lenght									: INT;					//		Długość chwytaka				| [mm]	(10-100)
	iCapSorterRobotProductDiametr								: INT;					//		Średnica nasadki				| [mm] 	(10-100)
	
//----------------------------------------CapSorterIntermediateTransporter---------------------------------------------------------------------------------------------------------------------------
	// Sorter nasadek, transporter zasypowy
	bCapSorterIntermediateTransporterEnableShow					: BOOL;					//		Aktywacja
	iCapSorterIntermediateTransporterAutoSpeedShow				: INT		:= 20;		//		Prędkość 					| [%] (1.0-100.0)
	iCapSorterIntermediateTransporterManualSpeedShow			: INT		:= 30;		//		Prędkość, manual 			| [%] (1.0-100.0)
	iCapSorterIntermediateTransporterEmptyingSpeedShow			: INT		:= 50;		//		Prędkość, opróżnianie 		| [%] (1.0-100.0)
	iCapSorterIntermediateTransporterDelayCountTimeShow			: INT		:= 100;		//		Timer pracy					| [ms]	(0.0-100_000.0)
	iCapSorterIntermediateTransporterReverseTimeShow			: INT		:= 4000;	//		Timer odwróconej pracy 		| [ms] (0.0-10_000.0)
	udiCapSorterIntermediateTransporterTimeProductOnSensorShow	: UDINT		:= 1800;	//		Czas produktu na czujniku 	| [ms] (0.0-10_000.0)	
	lrCapSorterIntermediateTransporterWheelAngleShow			: LREAL		:= 6;		//		Kąt zasypu 					| [°] (1.0-360.0)
	lrCapSorterIntermediateTransporterItemsSetValueShow			: LREAL	;				// 		Ilość detali na kołe		| []
	
//----------------------------------------CapSorterIntermediateBrush---------------------------------------------------------------------------------------------------------------------------
	//Sorter nasadek, szczotka transportera
	bCapSorterIntermediateBrushEnableShow						: BOOL;					//		Aktywacja
	iCapSorterIntermediateBrushAutoSpeedShow					: INT		:= 30;		//		Prędkość  					| [%] (0.0-100.0)
	iCapSorterIntermediateBrushManualSpeedShow					: INT		:= 30;		//		Prędkość, manual 			| [%] (0.0-100.0)
	iCapSorterIntermediateBrushEmptyingSpeedShow				: INT		:= 30;		//		Prędkość, opróżnianie 		| [%] (0.0-100.0)
	lrCapSorterIntermediateBrushPositionHeightSVShow			: LREAL		:= 45;		//		Wysokość 					| [mm] (0.0-10_000.0)

//----------------------------------------CapSorterBrush1OnWheel---------------------------------------------------------------------------------------------------------------------------
	// Sorter nasadek, szczotka stolu 1
	bCapSorterBrush1OnWheelEnableShow							: BOOL;					//		Aktywacja
	iCapSorterBrush1OnWheelAutoSpeedShow						: INT		:= 30;		//		Prędkość 					| [%] (0.0-100.0)
	iCapSorterBrush1OnWheelManualSpeedShow						: INT		:= 30;		//		Prędkość, manual 			| [%] (0.0-100.0)
	iCapSorterBrush1OnWheelEmptyingSpeedShow					: INT		:= 30;		//		Prędkość, opróżnianie 		| [%] (0.0-100.0)
	lrCapSorterBrush1OnWheelPositionHeightSVShow				: LREAL		:= 45;		//		Wysokość 					| [mm] (0.0-10_000.0)
	
//----------------------------------------CapSorterBrush2OnWheel----------------------------------------------------------------------------------
	// Sorter nasadek, szczotka stolu 2
	bCapSorterBrush2OnWheelEnableShow							: BOOL;					//		Aktywacja
	iCapSorterBrush2OnWheelAutoSpeedShow						: INT		:= 30;		//		Prędkość 					| [%] (0.0-100.0)
	iCapSorterBrush2OnWheelManualSpeedShow						: INT		:= 30;		//		Prędkość, manual 			| [%] (0.0-100.0)
	iCapSorterBrush2OnWheelEmptyingSpeedShow					: INT		:= 30;		//		Prędkość, opróżnianie 		| [%] (0.0-100.0)
	lrCapSorterBrush2OnWheelPositionHeightSVShow				: LREAL		:= 45;		//		Wysokość 					| [mm] (0.0-10_000.0)

//------------------------------------------CapFeeder-------------------------------------------------------------------------------------------------------------------------	
	// Sorter nasadek, 
	bCapSorterFeederEnableShow									: BOOL;					//		Aktywacjaa
	bCapSorterFeederEnableTubeError								: BOOL;					// 		Aktywacja błedu słomki
	lrCapSorterFeederMover1InputPositionShow					: LREAL;				//		Pozycja wkładania, wózek 1 	| [mm] (?-?)
	lrCapSorterFeederMover2InputPositionShow					: LREAL;				//		Pozycja wkładania, wózek 2 	| [mm] (?-?)
	lrCapSorterFeederMover1OutputPositionShow					: LREAL;				//		Pozycja wyjmowania, wózek 1 | [mm] (?-?)
	lrCapSorterFeederMover2OutputPositionShow					: LREAL;				//		Pozycja wyjmowania, wózek 2 | [mm] (?-?)
	lrCapSorterFeederSlotDistanceShow							: LREAL;				//		Offset wkładania			| [mm] (?-?)			Old-(Odstęp między pozycjami kładzenia)
	lrCapSorterFeederMoverSpeedShow								: LREAL;				//		Prędkość				 	| [%] (0.0-100.0)
	lrCapSorterFeederMoverAccelerationShow						: LREAL;				//		Przyspieszenie 				| [mm/s²] 
	lrCapSorterFeederMoveJerkShow								: LREAL;				//		Zryw						| [mm/s³]

//-------------------------------------------------------------------------------------------------------------------------------------------------------------------	
	//CapPreScrewer		
	bCapSorterPreScrewerEnableShow								: BOOL;					// 		Aktywacja
	bCapSorterPreScrewerPicker1EnableShow						: BOOL;					// 		Aktywacja	
	bCapSorterPreScrewerPicker2EnableShow						: BOOL;					// 		Aktywacja
	bCapSorterPreScrewerPicker3EnableShow						: BOOL;					// 		Aktywacja	
	bCapSorterPreScrewerPicker4EnableShow						: BOOL;					// 		Aktywacja
	//Oś Z
	lrCapSorterPreScrewerPickZPositionShow						: LREAL;				//		Wysokość pobierania						| [mm]	
	lrCapSorterPreScrewerCatcherReleseShow						: LREAL;				//		nie używamy Wysokość otwierania chwytaka nakrętek	| [mm]		
	lrCapSorterPreScrewerCapCatcherZPositionShow				: LREAL;				//		Wysokość zamykania nakrętkek			| [mm]
	lrCapSorterPreScrewerTopZPositionShow						: LREAL;				//		Pozycja górna ośi Z						| [mm] 	
	lrCapSorterPreScrewerCartesianCatchZPositionShow			: LREAL; 				//      Wait Position
	lrCapSorterPreScrewerStrawCatcherZPositionShow				: LREAL;				//		Wysokość otwierania łapaczy słomek		| [mm]	
	LrCapSorterPreScrewerCheckStrawCatcherActuatorZPosition		: LREAL;				//		Wysokość sparawdzania cofania łapaczy słomek	| [mm]	
	lrCapSorterPreScrewerScrewerStartZPositionShow				: LREAL;				//		Wysokość początku zakręcania			| [mm]	
	lrCapSorterPreScrewerGripperOpenPositionShow				: LREAL;				//		Pozycja otwierania chwytaka butelek 	| [mm]
	lrCapSorterPreScrewerPlaceZPositionShow						: LREAL;				//		Wysokość odkładania - koniec załapywania gwintu	| [mm] 

	lrCapSorterPreScrewerThreadPitchShow						: LREAL;				//		Skok gwintu 		| [mm]	
	lrCapSorterPreScrewerMultipleStartThreadShow				: LREAL;				//		Krotność gwintu
	lrCapSorterPreScrewerNumberOfThreadTurnsShow				: LREAL;				//		Ilość obrotów
  	
	//Wspólne ruchi	
	lrCapSorterPreScrewerBendingDistanceShow					: LREAL;				//		Odległość zaokrąglania ruchów 			| [mm]		
	lrCapSorterPreScrewerStrawInsertDistance					: LREAL;				//		Odległość wspólnego ruchu, prowadzenie słomki	| [mm]		
	//Oś x
	lrCapSorterPreScrewerPickXMover1PositionShow				: LREAL;				//		Pozycja osi poziomej do pobierania, wozek 1	| [mm]
	lrCapSorterPreScrewerPickXMover2PositionShow				: LREAL;				//		Pozycja osi poziomej do pobierania, wozek 2	| [mm]
	lrCapSorterPreScrewerPlaceXPositionShow						: LREAL;				//		Pozycja osi poziomej do odkładania			| [mm]
	//Oś zakręcania
	lrCapSorterPreScrewerScrewFindingShow						: LREAL;				//		Kąt szukania gwintu							| [°]
	lrCapSorterPreScrewerScrewDistanceShow						: LREAL;				//		Kąt zakręcania								| [°]
	//Prédkośći                                                                                                                         	
	lrCapSorterPreScrewerPickerSpeedShow						: LREAL;				//		Prędkość									| [%]   
	lrCapSorterPreScrewerPickerSpeedWhenScrewerShow				: LREAL;				//		Prędkość osi Z przy zakręcaniu				| [%]   
	lrCapSorterPreScrewerPickerAccelerationShow					: LREAL;				//		Przyspieszenie								| [mm/s²] 		
	lrCapSorterPreScrewerPickerJerkShow							: LREAL;				//		Zryw										| [mm/s³]
                                                                                                                                        	
	lrCapSorterPreScrewerCatcherSpeedShow						: LREAL;				//		Prędkość									| [mm/s] 
	lrCapSorterPreScrewerCatcherAccelerationShow				: LREAL;				//		Przyspieszenie								| [mm/s²] 	
	lrCapSorterPreScrewerCatcherJerkShow						: LREAL;				//		Zryw										| [mm/s³]	                                                                                                                                 	
	lrCapSorterPreScrewerScrewSpeedShow							: LREAL;				//		Prędkość zakręcania							| [mm/s]
	lrCapSorterPreScrewerScrewAccelerationShow					: LREAL;				//		Przyspieszenie zakręcania				| [mm/s²]
	lrCapSorterPreScrewerScrewJerkShow							: LREAL;				//		Zryw zakręcania							| [mm/s³]

	//Oś łapacza słomki	
	lrCapSorterPreScrewerCatcherCatchingPositionShow			: LREAL;				//		Pozycja łapania słomki					| [mm]
	lrCapSorterPreScrewerCatcherPlacePositionShow				: LREAL;				//		Pozycja dolna łapacza słomki			| [mm]
	lrCapSorterPreScrewerCatcherHightSVShow						: LREAL;				//		Nastawa wysokości stacji łapacza słomek		| [mm]
	//Kalibracja chwytaków butelki
	bCapSorterPreScrewerBottleCatcherEnableShow					: BOOL;					//		Actywacja chwytaków butelki
	lrCapSorterPreScrewerBottleCatch1OpenValueShow				: LREAL;				//		Chwytak 1 | wartość kalibracji otwartego chwytaka
	lrCapSorterPreScrewerBottleCatch1CloseValueShow				: LREAL;				//		Chwytak 1 | wartośc kalibracji zamkniętego chwytaka
	lrCapSorterPreScrewerBottleCatch2OpenValueShow				: LREAL;				//		Chwytak 2 | wartość kalibracji otwartego chwytaka
	lrCapSorterPreScrewerBottleCatch2CloseValueShow				: LREAL;				//		Chwytak 2 | wartość kalibracji zamkniętego chwytaka
	lrCapSorterPreScrewerBottleCatch3OpenValueShow				: LREAL;                //		Chwytak 3 | wartość kalibracji otwartego chwytaka
	lrCapSorterPreScrewerBottleCatch3CloseValueShow				: LREAL;				//		Chwytak 3 | wartość kalibracji zamkniętego chwytaka	
	lrCapSorterPreScrewerBottleCatch4OpenValueShow				: LREAL;                //		Chwytak 4 | wartość kalibracji otwartego chwytaka
	lrCapSorterPreScrewerBottleCatch4CloseValueShow				: LREAL;				//		Chwytak 4 | wartość kalibracji zamkniętego chwytaka
	                                                        	
	lrCapSorterPreScrewerBottleCatchToleranceValueShow			: LREAL;				//		Tolerancja chwytaków
	lrCapSorterPreScrewerCatchAngleOpenSV						: LREAL := 180.0;		//		[] Kąt puszczania centrowników
	
	lrCapSorterPreScrewerWaitInPlaceTimeShow					: LREAL	:= 50;			//		Czas zatrzymania w miejscu odłożenia 	| [ms]
	
	bCapSorterPreScrewerCatchAngleOpenEnaShow					: BOOL;					// 		Aktywacja puszczania centrowników po osiągnięciu zadanego kątu
	bCapSorterPreScrewerPoundedInCap							: BOOL;					// 		Wbijana nasadka
	
//Parametry do obliczeń 
	lrCapSorterBottleHightShow									: LREAL;				//		Wysokość butelki
	lrCapSorterBottleNeckHightShow								: LREAL;				// 		Wysokość szyjki butelki
	lrCapSorterCapHightShow										: LREAL;				// 		Wysokość zamknięcia
	lrCapSorterCapNeckHightShow									: LREAL;				//		Wysokość szyjki zamknięcia
	lrCapSorterPreScrewerCheckValveShow							: LREAL;				//		Długość zaworu zwrotnego				| [mm]
	
	lrCapSorterMoverHightShow									: LREAL := 226.0;		//		Wysokość wózków (Kartezjanem dotknąć ssawkami gniazdo do wkładania zamknięć)
	
//Rezerwa	
	lrCapSorterSpare1											: LREAL;				//Rezerwa 1
	lrCapSorterSpare2											: LREAL;				//Rezerwa 2
	lrCapSorterSpare3											: LREAL;				//Rezerwa 3
	lrCapSorterSpare4											: LREAL;				//Rezerwa 4
	lrCapSorterSpare5											: LREAL;				//Rezerwa 5
	lrCapSorterSpare6											: LREAL;				//Rezerwa 6
	lrCapSorterSpare7											: LREAL;				//Rezerwa 7	
	
	
	
END_VAR

// ---- GVLs/UVFF/GVL_UVFF.TcGVL
VAR_GLOBAL
	

	aCartesianYAxisRef										: AXIS_REF;
	aCartesianZAxisRef										: AXIS_REF;
	aPreScrewerAxisRef										: AXIS_REF;
	aCatcherAxisRef											: AXIS_REF;
	
	CapPreSrewerBottleCatch1Error							:S_Error;								// 1 Chwytak butelek 
	CapPreSrewerBottleCatch2Error							:S_Error;								// 2 Chwytak butelek

    lrCapPreSrewerBottleCatch1ClosedValue                    	:LREAL;                        // Chwytak 1 | wartość kalibracji zamkniętego chwytaka
    lrCapPreSrewerBottleCatch1OpenValue                      	:LREAL;                        // Chwytak 1 | wartość kalibracji otwartego chwytaka
    lrCapPreSrewerBottleCatch2ClosedValue                    	:LREAL;                        // Chwytak 2 | wartość kalibracji zamkniętego chwytaka
    lrCapPreSrewerBottleCatch2OpenValue                      	:LREAL;                        // Chwytak 2 | wartość kalibracji otwartego chwytaka
  
    lrCapPreSrewerBottleCatchTolerance                       	:LREAL;                        // Tolerancja szyjki butelki pod dozownikami [0-100%]      
	bSimulation													: BOOL;
	bSimpleSimulationLogic										: BOOL;
	
	
	ftVacuumSensor1												: F_TRIG;
	ftVacuumSensor2												: F_TRIG;
	ftVacuumSensor3												: F_TRIG;				
	ftVacuumSensor4                                             : F_TRIG;
	
	diTest1														: DINT;
	diTest2														: DINT;
	diTesy3														: DINT;
	diTest4														: DINT;
END_VAR

// ---- GVLs/UVFF/GVL_VIS.TcGVL
(*
Nazwa:			GVL_VIS
Opis:			Zmienne dla wizualizacji
Wersja:			v0.2
Data:			2024-02-20
Autor:			MK
Urzadzenia:		
Konfiguracja:	
Info:
Zmiany:
- 20240220 [DP] Poprawki przed nowa wizką
*)

{attribute 'qualified_only'}
VAR_GLOBAL
	(*Legenda dla wizki :
		[H] - Hidden, prawdopodobnie nie potrzebne
		[I] - Info, informacja,
		[L] - Later, do zrobienia później, być może do przerobienia
	Uprawienia:
		brak opisu - operator
		[m] - Meechanik i powyżej
		[t] - Technolog i powyżej
		[s] - Serwis i powyżek
		[a] - Admin			
	*)

//-----------------------------------------CapSorterWheel--------------------------------------------------------------------------------------------------------------------------	
	//Sorter nasadek, koło
	iCapSorterWheelState							: INT;				// Stan
	sCapSorterWheelState							: STRING;   		// Stan
	bCapSorterWheelHoming							: BOOL;             // Bazowanie					// Przycisk bistabilny                     Bazowanie                                       									
	bCapSorterWheelManualWheelRight    				: BOOL;   			// Do przodu					// Przycisk monostabilny                     						
	bCapSorterWheelManualWheelLeft     				: BOOL;  			// Do tyłu						// Przycisk monostabilny  						
	bCapSorterWheelManualContinuousMovement			: BOOL;				// obrót o zadany kąt			// Przycisk bistabilny					
                                                                                               
//-----------------------------------------CapSorterCamera--------------------------------------------------------------------------------------------------------------------------	
	//Sorter nasadek, system wizyjny
	iCapSorterCameraState							: INT;				// Stan
	sCapSorterCameraState							: STRING;			// Stan
	bCapSorterCameraHoming							: BOOL;				// Bazowanie					// Przycisk bistabilny    	                                                	
	bCapSorterCameraManualRun						: BOOL;				// Zrób zdięcie					// Przycisk monostabilny
	bCapSorterBacklightManualStart					: BOOL;				// Podświetlenie stolu			// Przycisk bistabilny  
	uiCapSorterCameraActualJobIDLoaded				: UDINT;   	        // Program załadowany			// Pole do wyświetlania wartości                                   
	lrCapSorterCameraPickPointXVisu					: LREAL;			// Współrzędne produktu, X		// Pole do wyświetlania wartości
	lrCapSorterCameraPickPointYVisu					: LREAL;			// Współrzędne produktu, Y		// Pole do wyświetlania wartości
	lrCapSorterCameraPickPointAngleVisu				: LREAL;			// Kąt produktu					// Pole do wyświetlania wartości
                                                 	
//------------------------------------------ CapSorterRobot-------------------------------------------------------------------------------------------------------------------------	
	//Sorter nasadek, robot
	iCapSorterRobotState							: INT;				// Stan
	sCapSorterRobotState							: STRING;           // Stan
	bCapSorterRobotHoming							: BOOL;             // Bazowanie					// Przycisk bistabilny                                	
	
	bCapSorterRobotManualVacumOn					: BOOL; 			// Ssawka						// Przycisk bistabilny
	bCapSorterRobotManualRejectOn					: BOOL;				//Odrzut						// Przycisk bistabilny
	bCapSorterRobotManualGripperArmPosition1		: BOOL;  			// Ramię robota					// Przycisk bistabilny	
	bCapSorterRobotReadyPosition 					: BOOL;     		// Gotowość                                                                  	
	bCapSorterRobotPreparePick 						: BOOL;     		// Przygotuj do pobrania	
	bCapSorterRobotPick 							: BOOL;     		// Pobierz						// Przycisk bistabilny
	bCapSorterRobotPreparePlace						: BOOL;     		// Przygotuj do odłożenia
	bCapSorterRobotPlace							: BOOL;     		// Odłóż						// Przycisk bistabilny
	diCapSorterRobotPlaceId							: DINT; 			// Slot odłożenia | (1-4) 		// Pole do wpisywania wartosci
	diCapSorterRobotSpeed							: DINT; 			// Prędkość | [%] (1-100)		// Pole do wpisywania wartosci

		
//----------------------------------CapSorterTransporter---------------------------------------------------------------------------------------------------------------------------------
	//Sorter nasadek, transporter zasobnika
	iCapSorterTransporterState						: INT;				// Stan
	sCapSorterTransporterState						: STRING;           // Stan
	bCapSorterTransporterHoming						: BOOL;		        // Bazowanie					// Przycisk bistabilny                                          	
	bCapSorterTransporterManualTankConveyor			: BOOL;       		// Do przodu					// Przycisk bistabilny
	bCapSorterTransporterManualTankConveyorRevers	: BOOL;             // Do tyłu						// Przycisk bistabilny                                   	                                           	
		
	
	
//----------------------------------------CapSorterIntermediateTransporter---------------------------------------------------------------------------------------------------------------------------	
	// Sorter nasadek, transporter zasypowy
	iCapSorterIntermediateTransporterState			: INT;				// Stan
	sCapSorterIntermediateTransporterState			: STRING;	        // Stan                                      
	bCapSorterIntermediateTransporterHoming			: BOOL;             // Bazowanie					// Przycisk bistabilny   
	bCapSorterIntermediateTransporterManualForward	: BOOL;             // Do przodu					// Przycisk bistabilny
	bCapSorterIntermediateTransporterManualBackward	: BOOL;				// Do tyłu						// Przycisk bistabilny   
	
//----------------------------------------CapSorterIntermediateBrush---------------------------------------------------------------------------------------------------------------------------	
	//Sorter nasadek, szczotka transportera
	iCapSorterIntermediateBrushState				: INT;	  			// Stan
	sCapSorterIntermediateBrushState				: STRING;           // Stan
	bCapSorterIntermediateBrushHoming				: BOOL;             // Bazowanie					// Przycisk bistabilny                                      
	bCapSorterIntermediateBrushWeightSet			: BOOL;				// Ustaw pozycje				// Przycisk bistabilny
	bCapSorterIntermediateBrushManualForward		: BOOL;             // Do przodu					// Przycisk bistabilny
	bCapSorterIntermediateBrushManualBackward		: BOOL;		        // Do tyłu						// Przycisk bistabilny                                           
	bCapSorterIntermediateBrushManualLiftUp			: BOOL;				// Do góry						// Przycisk monostabilny
	bCapSorterIntermediateBrushManualLiftDown		: BOOL;             // Do dołu						// Przycisk monostabilny
	lrCapSorterIntermediateBrushActualHeight		: LREAL;			//Aktualna wysokosc | [mm]				// Pole do wyświetlania wartości
		
//-------------------------------------------CapSorterBrush1------------------------------------------------------------------------------------------------------------------------
	// Sorter nasadek, szczotka stolu 1
	iCapSorterBrush1OnWheelState					: INT;				// Stan
	sCapSorterBrush1OnWheelState					: STRING;           // Stan
	bCapSorterBrush1OnWheelHoming					: BOOL;	            // Bazowanie					// Przycisk bistabilny                                                       
	bCapSorterBrush1WeightSet						: BOOL;				// Ustaw pozycje				// Przycisk bistabilny
	bCapSorterBrush1OnWheelManualLiftUp				: BOOL;             // Do przodu					// Przycisk bistabilny
	bCapSorterBrush1OnWheelManualLiftDown			: BOOL;	            // Do tyłu						// Przycisk bistabilny                                                       
	bCapSorterBrush1OnWheelManualDriveForward		: BOOL;             // Do góry						// Przycisk monostabilny
	bCapSorterBrush1OnWheelManualDriveBackward		: BOOL;             // Do dołu						// Przycisk monostabilny
	lrCapSorterBrush1OnWheelActualHeight			: LREAL;	        //Aktualna wysokosc | [mm]				// Pole do wyświetlania wartości
	
//----------------------------------------CapSorterBrush2---------------------------------------------------------------------------------------------------------------------------	
	// Sorter nasadek, szczotka stolu 2
	iCapSorterBrush2State							: INT;				// Stan
	sCapSorterBrush2State							: STRING;           // Stan
	bCapSorterBrush2Homing							: BOOL;	            // Bazowanie					// Przycisk bistabilny                   
	bCapSorterBrush2WeightSet						: BOOL;				// Ustaw pozycje				// Przycisk bistabilny	
	bCapSorterBrushManualBrush2OnWheelLiftUp		: BOOL;             // Do przodu					// Przycisk bistabilny
	bCapSorterBrushManualBrush2OnWheelLiftDown		: BOOL;             // Do tyłu						// Przycisk bistabilny                   
	bCapSorterBrushManualBrush2OnWheelDriveForward	: BOOL;             // Do góry						// Przycisk monostabilny
	bCapSorterBrushManualBrush2OnWheelDriveBackward	: BOOL;             // Do dołu						// Przycisk monostabilny
	lrCapSorterBrush2OnWheelActualHeight			: LREAL;            //Aktualna wysokosc | [mm]				// Pole do wyświetlania wartości		

//-------------------------------------------------------------------------------------------------------------------------------------------------------------------	
	//Sorter nasadek, CapFeeder
	iCapSorterFeederState							: INT;			// Stan
	lrCapSorterFeederMover1CVShow					: LREAL;		// Pozycja mówera 1
	lrCapSorterFeederMover2CVShow					: LREAL;		// Pozycja mówera 2  
	sCapSorterFeederState							: STRING;       // Stan
	bCapSorterFeederHoming							: BOOL;			// Bazowanie						// Przycisk bistabilny 
	bCapSorterFeederMover1Forvard 					: BOOL;			// Mover 1 +						// Przycisk monostabilny
	bCapSorterFeederMover1Backward					: BOOL;			// Mover 1 -						// Przycisk monostabilny
	bCapSorterFeederMover2Forvard 					: BOOL;			// Mover 2 +						// Przycisk monostabilny
	bCapSorterFeederMover2Backward					: BOOL;			// Mover 2 -						// Przycisk monostabilny
	bCapSorterFeederMover1ActuatorIn				: BOOL;			// Mover 1 Do przodu				// Przycisk bistabilny
	bCapSorterFeederMover1ActuatorOut				: BOOL;			// Mover 1 Do tyłu					// Przycisk bistabilny
	bCapSorterFeederMover1PickPos					: BOOL;			// Mover 1, pozycja pobrania		// przycisk monostabilny
	bCapSorterFeederMover1PlacePos					: BOOL;			// Mover 1, pozycja odkładania		// przycisk monostabilny
	bCapSorterFeederMover2PickPos					: BOOL;			// Mover 2, pozycja pobrania		// przycisk monostabilny
	bCapSorterFeederMover2PlacePos					: BOOL;			// Mover 2, pozycja odkładania		// przycisk monostabilny
	
//-------------------------------------------------------------------------------------------------------------------------------------------------------------------	
	//Sorter nasadek, CapPreScrewer	
	iCapSorterPreScrewerState							: INT;			// Stan
	sCapSorterPreScrewerState							: STRING;       // Stan
	lrCapSorterPreScrewerYAxisCVShow					: LREAL;		// Pozycja kartezjana oś Y
	lrCapSorterPreScrewerZAxisCVShow					: LREAL;		// Pozycja kartezjana oś Z
	lrCapSorterPreScrewerCAxisCVShow					: LREAL;		// Pozycja kartezjana oś C  
	bCapSorterPreScrewerHoming							: BOOL;			// Bazowanie					// Przycisk bistabilny 
	bCapSorterPreScrewerSetOffsetEncoderAxisZ			: BOOL;			// Ustaw offset encodera osi Z	//	Przycisk monostabilny
	bCapSorterPreScrewerPicker1Catch					: BOOL;			// Chwytak 1					// 	Przycisk bistabilny 
	bCapSorterPreScrewerPicker2Catch					: BOOL;			// Chwytak 2					// 	Przycisk bistabilny 
	bCapSorterPreScrewerPicker3Catch					: BOOL;			// Chwytak 3					// 	Przycisk bistabilny 
	bCapSorterPreScrewerPicker4Catch					: BOOL;			// Chwytak 4					// 	Przycisk bistabilny 
	bCapSorterPreScrewerPicker1Vacuum					: BOOL;			// Podsys 1						// 	Przycisk bistabilny 	
	bCapSorterPreScrewerPicker2Vacuum					: BOOL;			// Podsys 2						// 	Przycisk bistabilny 	
	bCapSorterPreScrewerPicker3Vacuum					: BOOL;			// Podsys 3						// 	Przycisk bistabilny 	
	bCapSorterPreScrewerPicker4Vacuum					: BOOL;			// Podsys 4						// 	Przycisk bistabilny 	
	bCapSorterPreScrewerPicker1Reject					: BOOL;			// Oddmuch 1					// 	Przycisk bistabilny	
	bCapSorterPreScrewerPicker2Reject					: BOOL;			// Oddmuch 2					// 	Przycisk bistabilny	
	bCapSorterPreScrewerPicker3Reject					: BOOL;			// Oddmuch 3					// 	Przycisk bistabilny	
	bCapSorterPreScrewerPicker4Reject					: BOOL;			// Oddmuch 4					// 	Przycisk bistabilny	
	
		//Kartezjan
	bCapSorterPreScrewerCartesianYForward				: BOOL;			// Y +							// Przycisk monostabilny
	bCapSorterPreScrewerCartesianYBackward				: BOOL;			// Y -							// Przycisk monostabilny
	bCapSorterPreScrewerCartesianZForward				: BOOL;			// Z +							// Przycisk monostabilny
	bCapSorterPreScrewerCartesianZBackward				: BOOL;			// Z -							// Przycisk monostabilny
	bCapSorterPreScrewerCartesianCForward				: BOOL;			// C +							// Przycisk monostabilny
	bCapSorterPreScrewerCartesianCBackward				: BOOL;			// C -							// Przycisk monostabilny
	                                                    	        	
		//Łapacz słomki    
 	lrCapSorterPreScrewerStrawCatcherCVShow				: LREAL;		// Pozycja łapacza słomek                           	
    bCapSorterPreScrewerStrawCatcherUp					: BOOL;			// Chwytaki do góry 			// Przycisk monostabilny
	bCapSorterPreScrewerStrawCatcherDown				: BOOL;			// Chwytaki do dołu 			// Przycisk monostabilny	
	bCapSorterPreScrewerStrawCatcherCatchOpen			: BOOL;			// Otwórz chwytaki słomek		// Przycisk bistabilny
	bCapSorterPreScrewerStrawCatcherCatchClose			: BOOL;			// Zamknij chwytaki słomek		// Przycisk bistabilny
	bCapSorterPreScrewerStrawCatcherActuatorIn			: BOOL;			//  Wsuń łapacz słomek			// Przycisk bistabilny
	bCapSorterPreScrewerStrawCatcherActuatorOut			: BOOL;			//  Wysuń łapacz słomek			// Przycisk bistabilny
                                                    	

                                                		
		//Podnośnik stacji wkladania nakrętek       		            	 
	bCapSorterPreScrewerCatcherStationUp					: BOOL;			// Stacja do góry 				// Przycisk monostabilny
	bCapSorterPreScrewerCatcherStationDown					: BOOL;			// Stacja do dołu 				// Przycisk monostabilny                 			
	bCapSorterPreScrewerBottleCatcherCatch					: BOOL;			// Chwytaki Butelek				// Przycisk bistabilny	
	lrCapSorterPreScrewerCatcherStationHeightCV				: LREAL;		// Aktualna wysokość chwytaka
	bCapSorterPreScrewerCatcherStationHeightSet				: BOOL;			// Ustaw pozycje				// Przycisk bistabilny
	bCapSorterPreScrewerBottleCatchOpenCalibration			: BOOL;			// Kalibruj otwarcie			// Przycisk bistabilny
	bCapSorterPreScrewerBottleCatchCloseCalibration			: BOOL;			// Kalibruj zamknięcie			// Przycisk bistabilny
	bCapSorterPreScrewerNextStep							: BOOL;			// Kolejny krok w serwice mode
                                                                        
	//Chwytak szyjki butelki pod wkladaczem nakrentek 1234                  
	bCapSorterPreScrewerCatchStationHoming	      			: BOOL;			// [H] Homing  					// Przycisk bistabilny	
	lrCapSorterPreScrewerCatchStationHeightSVShow			: LREAL;  		// Pozycja chwytaka
	bCapSorterPreScrewerManualBottleCatcherCatch			: BOOL;											// Przycisk bistabilny	        
 	
	
	bCapSorterManualVacuumPump								: BOOL; 
	// 1-Fliptop (prosta scieżka), 2-Pompka/Atomizer (Stawianie do pionu), 3-Fliptop z boku (stawianie do pionu + detekcja obróconej)
	AsCapSorterProductType									: ARRAY [1..10] OF STRING;
//	iCapSorterProductType									: INT;
	//
	AsCapSorterIndexShow									: ARRAY [1..30] OF STRING;	
//	uiCapSorterIndexShow									: UDINT;
	

	bCapSorterFeederAdvancedHoming							: BOOL;			// Bazowanie wózków "na zderzak"	
	bCapSorterPreScrewerAdvancedHoming						: BOOL;			// Bazowanie zaawansowane dotyczy osi Y
	
	lrCapSorterPreScrewerVacuumLevel_1						: LREAL;			// Podcisnienie na głowicy nr1	[Bar]
	lrCapSorterPreScrewerVacuumLevel_2						: LREAL;			// Podcisnienie na głowicy nr2	[Bar]
	lrCapSorterPreScrewerVacuumLevel_3						: LREAL;			// Podcisnienie na głowicy nr3	[Bar]
	lrCapSorterPreScrewerVacuumLevel_4						: LREAL;			// Podcisnienie na głowicy nr4	[Bar]	
	
//-----------------------------------------------------------------------------------------------------------------------------------------------------

	bCapSorterCalculateParameters							: BOOL;			//	Oblicz paramaretry maszyny	//przycisk monostabilny
	bCapSorterSpare1										: BOOL;			//Rezerwa 1
	bCapSorterSpare2										: BOOL;			//Rezerwa 2
	bCapSorterSpare3										: BOOL;			//Rezerwa 3
	bCapSorterSpare4										: BOOL;			//Rezerwa 4
	bCapSorterSpare5										: BOOL;			//Rezerwa 5
	bCapSorterSpare6										: BOOL;			//Rezerwa 6
	bCapSorterSpare7										: BOOL;			//Rezerwa 7
	
	fbAlarms :FB_Events; 	//ActiveAlarms
	
	
END_VAR

// ---- GVLs/VIS.TcGVL
(*
Nazwa:			VIS
Opis:			Zmienne wykorzystywane i zmieniane tylko z wizualizacji
Wersja:			v0.2
Data:			2024-02-06
Autor:			DP,MP
Urzadzenia:		
Konfiguracja:	
Info:
Zmiany:
- 20240205 [DP] Poprawki przed nowa wizką
*)

{attribute 'qualified_only'}

VAR_GLOBAL	
	
(********DANE MASZYNY***********)
sType: STRING[255];
sSerialNumber: STRING[255];
rProgramVersion: REAL;
rLastTimeChanges: REAL;
(*******************************)	

    (* OPISY ZMIENNYCH TYPU INT DO POŚWWIETLANIA STANÓW STACJI
	E_PackMLState : 
					eUndefined				:=  0, //----Nieużywany
					eClearing 				:=  1, //----Nieużywany
					eStopped 				:=  2, //Błąd
					eStarting 				:=  3, //Uruchamianie
					eIdle 					:=  4, //Postój
					eSuspended 				:=  5, //---Nieużywany
					eExecute 				:=  6, //Praca
					eStopping	 			:=  7, //Zatrzymywanie
					eAborting 				:=  8, //Zatrzymywanie awaryjne
					eAborted 				:=  9, //Zatrzymano awaryjnie
					eHolding 				:= 10, //---Nieużywany
					eHeld 					:= 11, //---Nieużywany
					eUnholding 				:= 12, //---Nieużywany
					eSuspending 			:= 13, //---Nieużywany
					eUnsuspending 			:= 14, //---Nieużywany
					eResetting 				:= 15, //Resetowanie błędu, bazowanie
					eCompleting 			:= 16, //---Nieużywany
					eComplete	 			:= 17  //---Nieużywany
	
	E_Station :
					eDisabled 				:= 0, // Stan nieaktywnosci (Stacja wyłączona)             
					eAborted 				:= 1, // Stan bezpiecznego zatrzymania (po Abortingu) 
					eAborting 				:= 2, // Stan bezpiecznego zatrzymywania (po EStopie)
					eError 					:= 3, // Stan błędu 		
					eResetting 				:= 4, // Stan resetowania bledu (po Errorze)		                
					eManualMovement 		:= 5, // Stan ruchów manualnych         
					eHoming 				:= 6, // Stan bazowania 
					eHomingDone 			:= 7, // Stan wykonania bazowania 
					ePreparingToReady 		:= 8, // Stan przygotowywania do gotowosci (zawsze przed Ready)           
					ePreparingToDisable 	:= 9, // Stan przygotowywania do nieaktywnosci (po wyłączeniu Enable)                               
					eReady					:= 10,// Stan gotowosci 
					eStopping 				:= 11,// Stan zatrzymywania 
					eStarting 				:= 12,// Stan uruchamiania (po Ready)
					eRunning 				:= 13 // Stan wykonywania cyklu (po Startingu), w tym stanie osobny 
					
					
	Legenda dla wizki :
	[H] - Hidden, prawdopodobnie nie potrzebne
	[I] - Info, informacja,
	[L] - Later, do zrobienia później, być może do przerobienia
	Uprawienia:
	brak opisu - operator
	[m] - Meechanik i powyżej
	[t] - Technolog i powyżej
	[s] - Serwis i powyżek
	[a] - Admin			
	*)
	(*****Zmienne ogólne****)
	
	(* Wykresy dozowania*)
	aPoints												: ARRAY [0..11,0..599] OF ST_Point;	// Sam wykres wybrando doziwniki + jego simulacji
	udiDossagerNum										: UDINT	:=	0;						// Wybrany dozownik 0 - pierwszy, 3 - czwarty
	bDrawChart											: BOOL;								// Cykl simulacji
	nDrawLenght										:INT;
	nTimeMarkerDSPh1                                :INT;
	nTimeMarkerDSPh2                                :INT;
	nTimeMarkerDSPh3                                :INT;
	nTimeMarkerDSPh4								:INT;
	nTimeMarkerDSPh5								:INT;
	aHorizontalChart								: ARRAY[0..4] OF ARRAY [0..0] OF INT;
	lrTorqMin										:LREAL;
	lrTorqMax										:LREAL;
	aWeightPoints									: ARRAY [0..7,0..9999] OF ST_Point_1;
	
	
	
	
	
	
	
	
	//Zmienne przejść do różnych stanów	
	iMachineState										:UINT;						// Stan maszyny
	sMachineState										:STRING; 					// Stan maszyny
	wsMachineState										:WSTRING; 					// Stan maszyny

	//Okno przezbrajania po wyborze receptury
	bMachinePartsChangeOver								:BOOL;						// Włączone przezbrajanie (ustawić z wizki)
	iMachinePartsChangeOver								:INT;						// Stan przezbrajania (0-ruch,1-pozycja gorna,-1-pozycja dolna) 
	bBottleSorterDisable								:BOOL:=FALSE;				// Wyłączenie sortera butelek
	bCapSorterDisable									:BOOL:=FALSE;				// Wyłączenie sortera nasadek
	
	//Ekran z komunikatami
	bDialogBoxOn										:BOOL;		 				// Wyświetl okno komunikatów
	bDialogBoxText										:STRING[255];				// Treść na oknie komunikatów 
	bDialogBoxText2										:STRING[255];				// Treść na oknie komunikatów (nie tłumaczone, zmienne)
	sDialogBoxPicture									:STRING[255];				// Nazwa obrazka który ma sie wyświetlać, '' - brak obrazu, 1,2,ok,info,uwaga 
																					// (odnosi się do pliku pictures.txt gdzie są podaje lokalizacje obrazków)
																					(*	[{"ImagePath":"c:\\img\\img1.png","ImageID":"1"}, 
																						{"ImagePath":"c:\\img\\img2.png","ImageID":"2"},
																						{"ImagePath":"c:\\img\\ok.png","ImageID":"ok"},
																						{"ImagePath":"c:\\img\\info.png","ImageID":"info"},
																						{"ImagePath":"c:\\img\\uwaga.png","ImageID":"uwaga"}] *)
	bDialogBoxAck										:BOOL;						// Przycisk OK
	bDialogBoxCancelAck									:BOOL;						// Przycisk ANULUJ
	nDialogBoxType										:UINT;						// Rodzaj okna, 0-nic, 1-tylko przycisk OK, 2 - tylko przycisk Anuluj, 3 - Przycisk OK i Anuluj
	bDialogBoxAckNeeded									:BOOL;						// [H] Potrzebne potwierdzenie					

	wsDialogBoxText										:WSTRING;				// Treść na oknie komunikatów 
	wsDialogBoxText2									:WSTRING;				// Treść na oknie komunikatów (nie tłumaczone, zmienne)
	
	//Wyświetlanie informacji na ekranie głównym
	//Przyczyny odrzuceń (wyświetlić na ekranie głównym bez dodatkowego odpisu)
	sBadPackageReason1									:STRING;					// Powód odrzutu butelek 		//sBadPackageReason1 sBadPackageReason1
	sBadPackageReason2									:STRING;					//								//sBadPackageReason2 sBadPackageReason2
	sBadPackageReason3									:STRING;					//								//sBadPackageReason3 sBadPackageReason3	
	iBadPackageReasonCount1								:INT;						// Ilość odrzuconych opakowań
	iBadPackageReasonCount2								:INT;						//
	iBadPackageReasonCount3								:INT;						//
	wsBadPackageReason1									:WSTRING;					// Powód odrzutu butelek 		//sBadPackageReason1 sBadPackageReason1
	wsBadPackageReason2									:WSTRING;					//								//sBadPackageReason2 sBadPackageReason2
	wsBadPackageReason3									:WSTRING;					//								//sBadPackageReason3 sBadPackageReason3	
	AStBadPackageReason									:ARRAY[0..63] OF S_Information;	// ID informacji do powodów odrzuceń
	bBadPackageReasonReset								:BOOL;						// Czyszczenie tablicy odrzuceń
	
	iNumbersOfFormsBetweenWeightAndScrewers				:INT;						// Ilość formatek pomiędzy wagą a zakręcarkami: zmienna
	
	sSlowestStation1									:STRING;					//	Najwolniejsza stacja nr 1	//sSlowestStation1 iSlowestStationCount1
	sSlowestStation2									:STRING;					//	Najwolniejsza stacja nr 2	//sSlowestStation2 iSlowestStationCount2
	sSlowestStation3									:STRING;					//	Najwolniejsza stacja nr 3	//itd.
	sSlowestStation4									:STRING;					//	Najwolniejsza stacja nr 4
	sSlowestStation5									:STRING;					//	Najwolniejsza stacja nr 5	
	iSlowestStationCount1								:INT;					  	//	Czas cyklu dla najwolniejszej stacji nr 1
	iSlowestStationCount2								:INT;					  	//	Czas cyklu dla najwolniejszej stacji nr 2
	iSlowestStationCount3								:INT;					  	//	Czas cyklu dla najwolniejszej stacji nr 3
	iSlowestStationCount4								:INT;					  	//	Czas cyklu dla najwolniejszej stacji nr 4
	iSlowestStationCount5								:INT;					  	//	Czas cyklu dla najwolniejszej stacji nr 5
	wsSlowestStation1									:WSTRING;					//	Najwolniejsza stacja nr 1	//sSlowestStation1 iSlowestStationCount1
	wsSlowestStation2									:WSTRING;					//	Najwolniejsza stacja nr 2	//sSlowestStation2 iSlowestStationCount2	
	wsSlowestStation3									:WSTRING;					//	Najwolniejsza stacja nr 3	//itd.	
	wsSlowestStation4									:WSTRING;					//	Najwolniejsza stacja nr 4	
	wsSlowestStation5									:WSTRING;					//	Najwolniejsza stacja nr 5	
	
	//Przyciski główne na HMI (wysuwany pasek lub na ekranie głównym)
	bDoorsUnlock										:BOOL;						// Otwórz drzwi 	
	bCycleReset											:BOOL;						// Reset cyklu 
	bCounterReset										:BOOL;						// Reset Liczników
	bConfectionEnding									:BOOL; 						// Zakończenie konfekcji
	bWeighingForm										:BOOL;						// [m] Przeważanie formatek
	bCapSorterEmptyingMode								:BOOL;						// Opróżnianie sortera nakrętek
	bBottleSorterEmptyingMode							:BOOL;						// Opróżnianie sortera butelek
	bBottleDeleteUnderDispencers						:BOOL;						// Usuń butelki pod dozownikami
	bSingleRealeseIfNoCapFromScrewers					:BOOL:=FALSE;						// Wypuszczanie pojedyńczo z zakręcarek jeżeli nie ma nasadki
	
	//Zmienne wystawiane z HMI
	bServiceMode										:BOOL; 						// Tryb serwisowy 
	bSimulation											:BOOL;						// [s] Przycisk trybu symulacyjnego
	bCheckStart 										:BOOL;						// Próba uruchomienia (PLC ustawia na 1, HMI na 0)
	bAllowStart 										:BOOL;						// Uruchomienie maszyny możliwe (HMI ustawia na 1 po bCheckStart i ktoś jest zalogowany, PLC ustawia na 0)
	iHMICommunication									:INT;						// [I] Licznik komunikacji, gdy się nie zmienia przez jakiś czas, wizka może wystawiać błąd
	bRecipeCalculate									:BOOL;						// Oblicz parametry receptury

	//[s] Zmienne tylko dla serwisu
	bWritePersistent									:BOOL; 						// [H] Zmienna zapisujaca wartosci zmiennych persistent
	bCycleStart											:BOOL;	(**)				// [H] Zdalny start/stop maszyny
	
	//Liczniki 
	uiCounterMachineEfficiency							:UINT; 						// Wydajność chwilowa maszyny[szt./h]
	uiCounterInstantEfficiency							:UINT; 						// Wydajność chwilowa prawidłowych butelek [szt./h]
	uiCounterAverageEfficiency							:UINT;						// Średnia wydajność [szt./h]
	udiCounterShiftBottles								:UDINT;						// Zmianowa ilość butelek [szt.]					
	uiCounterGoodBottles								:UINT;						// Prawidłowo napełnione opakowania [szt.]
	uiCounterBadBottles									:UINT;						// Odrzucone opakowania [szt]
	//Liczniki OEE
	udiCounterExecuteTime								:UINT;						// Cza pracy [min]
	udiCounterReadyTime									:UINT;						// Cza postoju [min]
	udiCounterErrorTime									:UINT;						// Cza błędu [min]
	
	//Lampki w trybie serwisowym pomocne do ustawiania stacji
	bCapPuttedCheckSensor								:BOOL;						// Czujnik nasadki przed zakręcarką
	bCapCorrectCheckCapOnSensor							:BOOL;						// Czujnik nasadki za zakręcarką
	bCapCorrectCheckCapNotScrewedSensor					:BOOL;						// Czujnik źle zakręconej nasadki

	(*Wykresy, statystyki, informacje*) 
	//Pomiary wag i dozowań do wyświetlenia na ekranie głównym
	lrDispencer1DoseVolumeCV							:LREAL;						// Doza 1 [ml]
	lrDispencer2DoseVolumeCV							:LREAL;						// Doza 2 [ml]
	lrDispencer3DoseVolumeCV							:LREAL;						// Doza 3 [ml]	
	lrDispencer4DoseVolumeCV							:LREAL;						// Doza 4 [ml]	
	lrDispencer1WeightMeasured							:LREAL;						// Waga z dozownika 1 [g]	
	lrDispencer2WeightMeasured							:LREAL;						// Waga z dozownika 2 [g]		
	lrDispencer3WeightMeasured							:LREAL;						// Waga z dozownika 3 [g]	
	lrDispencer4WeightMeasured							:LREAL;						// Waga z dozownika 4 [g]	
	bDispencer1WeightMeasured							:BOOL;						// [H] Waga zmierzona z dozownika nr 1	
	bDispencer2WeightMeasured							:BOOL;						// [H] Waga zmierzona z dozownika nr 2
	bDispencer3WeightMeasured							:BOOL;						// [H] Waga zmierzona z dozownika nr 3
	bDispencer4WeightMeasured							:BOOL;						// [H] Waga zmierzona z dozownika nr 4
		
	AsChartDose1										:ARRAY [0..500] OF STRING;	// [L] Wykres ostatniego dozowania 1 "Czas;PozycjaTłoka;PozycjaPodnośnika;ZawórSsący;ZaworDozujacy;Tacka" 
	AsChartDose2										:ARRAY [0..500] OF STRING;	// [L] Wykres ostatniego dozowania 2 "Czas;PozycjaTłoka;PozycjaPodnośnika;ZawórSsący;ZaworDozujacy;Tacka" 									
	AsChartDose3										:ARRAY [0..500] OF STRING;	// [L] Wykres ostatniego dozowania 3 "Czas;PozycjaTłoka;PozycjaPodnośnika;ZawórSsący;ZaworDozujacy;Tacka" 									
	AsChartDose4										:ARRAY [0..500] OF STRING;	// [L] Wykres ostatniego dozowania 4 "Czas;PozycjaTłoka;PozycjaPodnośnika;ZawórSsący;ZaworDozujacy;Tacka" 			
	AStAsChartDose1										:ARRAY [0..100] OF ARRAY [0..5,0..500] OF INT; // [L] Wykres ostatniego dozowania 1 "Czas;PozycjaTłoka;PozycjaPodnośnika;ZawórSsący;ZaworDozujacy;Tacka"
	AStAsChartDose2										:ARRAY [0..100] OF ARRAY [0..5,0..500] OF INT; // [L] Wykres ostatniego dozowania 1 "Czas;PozycjaTłoka;PozycjaPodnośnika;ZawórSsący;ZaworDozujacy;Tacka"
	AStAsChartDose3										:ARRAY [0..100] OF ARRAY [0..5,0..500] OF INT; // [L] Wykres ostatniego dozowania 1 "Czas;PozycjaTłoka;PozycjaPodnośnika;ZawórSsący;ZaworDozujacy;Tacka"
	AStAsChartDose4										:ARRAY [0..100] OF ARRAY [0..5,0..500] OF INT; // [L] Wykres ostatniego dozowania 1 "Czas;PozycjaTłoka;PozycjaPodnośnika;ZawórSsący;ZaworDozujacy;Tacka"
	
	
	AsChartGripperScrewer1								:ARRAY [0..500] OF STRING;	// [L] Wykres ostatniego zakręcania 1 "Czas;Wysokość;Obrót;Moment;SiłownikChwytania;;" 
	AsChartGripperScrewer2								:ARRAY [0..500] OF STRING;	// [L] Wykres ostatniego zakręcania 2 "Czas;Wysokość;Obrót;Moment;SiłownikChwytania;;" 
	AStChartGripperScrewer1								:ARRAY [0..100] OF ARRAY [0..5,0..500] OF INT;	// [L] Wykres ostatniego zakręcania 1 "Wysokość;Obrót;Prędkość;SiłownikChwytania;Czas;Pusty;;" 	
	AStChartGripperScrewer2								:ARRAY [0..100] OF ARRAY [0..5,0..500] OF INT;	// [L] Wykres ostatniego zakręcania 2 "Wysokość;Obrót;Prędkość;SiłownikChwytania;Czas;Pusty;;" 
	
	//[L] Przepisanie stanów wyjść ze sterownika na zmienne do HMI													
	//Pomiary przebiegu dozowania dozownika 1
	bHMIDispencer1SuckingValveActuator					:BOOL;						// Stan zaworu ssania dozownika nr 1
	bHMIDispencer1DosingValveActuator					:BOOL;						// Stan dozowania dozownika nr 1
	bHMIDispencer1DropCatcherValveActuator				:BOOL;						// Stan tacki dozownika nr 1
	//Pomiary przebiegu dozowania dozownika 2
	bHMIDispencer2SuckingValveActuator					:BOOL;						// Stan zaworu ssania dozownika nr 2
	bHMIDispencer2DosingValveActuator					:BOOL;						// Stan dozowania dozownika nr 2
	bHMIDispencer2DropCatcherValveActuator				:BOOL;						// Stan tacki dozownika nr 2
	//Pomiary przebiegu dozowania dozownika 3
	bHMIDispencer3SuckingValveActuator					:BOOL;						// Stan zaworu ssania dozownika nr 3
	bHMIDispencer3DosingValveActuator					:BOOL;						// Stan dozowania dozownika nr 3
	bHMIDispencer3DropCatcherValveActuator				:BOOL;						// Stan tacki dozownika nr 3
	//Pomiary przebiegu dozowania dozownika 4
	bHMIDispencer4SuckingValveActuator					:BOOL;						// Stan zaworu ssania dozownika nr 4
	bHMIDispencer4DosingValveActuator					:BOOL;						// Stan dozowania dozownika nr 4
	bHMIDispencer4DropCatcherValveActuator				:BOOL;						// Stan tacki dozownika nr 4
	//Prędkość podnośnika
	iHMIDispencersLifterMaxSpeed						:INT;						// Prędkość maksymalna podnośników dozowników (do ustawiania wykresów dozowników)

	//Tablica rejestrów z opisami
	AbFormPresent										:ARRAY [1..100] OF BOOL;	// Widoczność formatki formatki (np. .[2]=TRUE to formatka jest widoczna na 2 miejscu
	AsFormDescription									:ARRAY [1..100] OF STRING;	// Opis formatki (jedna literka, np. B,P,C) (.[2] to opis formatki na 2 miejscu)	
	                                        	
	(*****P00_Alarms***)    	                   									// Wyświetla tylko jeden błąd na raz, zatrzymuje maszynę    		                            	
	bErrorOccure										:BOOL:=FALSE;				// Błąd
	sStationInError										:STRING:='';				// Nazwa stacji
	udiStationInError									:UDINT:=0;					// ID Nazwa stacji która jest w stanie błędu 	//sStationName.xlsx
	udiStationErrorCode									:UDINT:=0;					// ID Kod błędu stacji							//sErrorString.xlsx
	sStationErrorDescription							:STRING(200):='';			// Opis błędu stacji - tłumaczony
	sStationErrorDescription2							:STRING(200):='';			// Opis błędu stacji - nie tłumaczony                    	
	bResetErrorVisuCmd									:BOOL:=FALSE;				// Reset błędu
	
	wsStationInError									:WSTRING:="";				// Nazwa stacji
	wsStationErrorDescription							:WSTRING(200):="";			// Opis 
	wsStationErrorDescription2							:WSTRING(200):="";			// Opis błędu (nie tłumaczony, zmienny)                      	

	fbAlarms 											:FB_Events;					// EventLogger

	//Warningi											// Wyświetlanie warningów, nie zatrzymuje maszyny	
	bWarningAcknowledgeAll								:BOOL;					 	// Przycisk potwierdzenia wszystkie ostrzeżenia
	bWarningNew											:BOOL;					 	// Pojawiło się nowe ostrzezenie 1s
	uliWarningOccure 									:ULINT;					 	// Wystąpienie ostrzezenia (każdy bit to inne ostrzeżenie [0..63])
	uliWarningAcknowledge 								:ULINT;						// Potwierdzenie ostrzezenia (każdy bit to inne ostrzeżenie [0..63])
	AsWarningDescription								:ARRAY [0..63] OF STRING;	// Opis ostrzeżenia (tablica na stałe wypisana)
															// VIS.AsWarningDescription[0]:='Niski pozom zbiornika nr 1';
															// VIS.AsWarningDescription[1]:='Niski pozom zbiornika nr 2';
															// VIS.AsWarningDescription[2]:='Zapełniony transproter odrzuconych opakowań';	
															// VIS.AsWarningDescription[3]:='			';
															// VIS.AsWarningDescription[4]:='Brak stabilizacji wagi przy pomiarach';
															// VIS.AsWarningDescription[5]:='Smarowanie robota';
															// VIS.AsWarningDescription[6]:='Brak odczytu RFID przed dozownikami';
															// VIS.AsWarningDescription[7]:='Brak odczytu RFID przed wagą';
															// VIS.AsWarningDescription[8]:='Brak odczytu RFID przed zakręcarką';
															// VIS.AsWarningDescription[9]:='Brak odczytu RFID pod robotem';

															// VIS.AsWarningDescription[10]:='Nieskalibrowany czujnik chwytaka szyjek pod dozownikami';
															// VIS.AsWarningDescription[11]:='Chwytak dozownika 1 - butelka nieprawidłowo chwycona';																					
															// VIS.AsWarningDescription[12]:='Chwytak dozownika 2 - butelka nieprawidłowo chwycona';																							
															// VIS.AsWarningDescription[13]:='Chwytak dozownika 3 - butelka nieprawidłowo chwycona';																							
															// VIS.AsWarningDescription[14]:='Chwytak dozownika 4 - butelka nieprawidłowo chwycona';	
															
															// VIS.AsWarningDescription[15]:='Zakręcarka 1 - przekroczenie czasu zakręcania - zmień ust.';		
															// VIS.AsWarningDescription[16]:='Zakręcarka 1 - przekroczenie czasu szukania gwintu - zmień ust.';
															// VIS.AsWarningDescription[17]:='Zakręcarka 1 - przekroczenie poślizgu - zmień ust.';
															// VIS.AsWarningDescription[18]:='Zakręcarka 1 - zbyt niska pozycja przy zakrecaniu - zmień ust.';
															// VIS.AsWarningDescription[19]:='Zakręcarka 2 - przekroczenie czasu zakręcania - zmień ust.';		
															// VIS.AsWarningDescription[20]:='Zakręcarka 2 - przekroczenie czasu szukania gwintu - zmień ust.';
															// VIS.AsWarningDescription[21]:='Zakręcarka 2 - przekroczenie poślizgu - zmień ust.';
															// VIS.AsWarningDescription[22]:='Zakręcarka 2 - zbyt niska pozycja przy zakrecaniu - zmień ust.';
															
	AwsActiveWarningDescription								:ARRAY [0..63] OF WSTRING;	//  Aktywne ostrzeżenia
	iActiveWarning											:INT;	// Ilość aktywnych ostrzeżeń				
	AudiActiveWarningDescriptionID							:ARRAY [0..63] OF UDINT;	// ID warningów do tłumaczeń na wizualizacji
																
	//Informacje // Pojawiają się na ekranie głównym i same znikają, jeżeli [0] > '' to wyświetl i usuń jak jest ''
	bInformationNew											:BOOL;					 		// Pojawiła sie nowa informacja
	AsInformationDescription  								:ARRAY[0..63] OF STRING; 		// Opis informacji, tablica na stałe wypisana
	iActiveInformation										:INT;					 		// Ilość aktywnych informacji
	AStInformationDescription								:ARRAY[0..63] OF S_Information;	// ID informacji do tłumaczeń na wizualizacji Struktura


																			
	(****P00_OEE*****) //Generowanie informacji do stworzenia OEE na wizualizacji
	// [L] Symbole według DescriptionStations.txt
	AsOEECycleTimes										:ARRAY [1..64] OF STRING;	// [L] Tabela czasów cykli 		[symbol_stacji;czas_w_ms] 	
	// Symbole według DecriptionRejectReason.txt
	// [L] Po ustawieniu powodu, dodawany jest ID
	sOEERejectionReason									:STRING;					// [L] Powód odrzuceń			[symbol_odrzucenia]

	sOEEText1											:STRING;					// Tekst 1			[PRACA:2h30MIN]
	sOEEText2											:STRING;					// Tekst 2			[POSTÓJ:1h30MIN]
	sOEEText3											:STRING;					// Tekst 1			[BŁĄD:2h30MIN]
	bOEEGenRaport										:BOOL;						//
	iOEEPackMLSuspendedReason							:INT;																																																																                                                        
	(**P01_BottleSorter***)
	// Sorter butelek
	bBottleSorterHold									:BOOL;
	// Zmienne czytane z innegro sterownika
	
	(***P01_BottleSorter***)
	// Podajnik butelek 
	iBottleFeederState									:INT;						// Stan
	sBottleFeederState									:STRING;					// Stan
	bBottleFeederRun									:BOOL;						// Cykl
	bBottleFeederHoming									:BOOL;						// Bazowanie 
	bBottleFeederIgnoreError							:BOOL;						// Ignoruj błędy
	bBottleFeederManualArmDown							:BOOL;						// Dół
	bBottleFeederManualArmLeft							:BOOL;						// Lewo
	bBottleFeederManualGate1							:BOOL;						// Szlaban 1 - lewy
	bBottleFeederManualGate2							:BOOL;						// Szlaban 2 - prawy
	bBottleFeederManualGripper							:BOOL;						// Chwytak
	bBottleFeederManualFormPositioning					:BOOL;						// Pozycjonowanie formatki
	bBottleFeederManualFormGate							:BOOL;						// Szlaban formatki		

	// Podajnik butelek - stół							
	iBottleFeederTurnTableState							:INT; 					 	// Stan
	sBottleFeederTurnTableState							:STRING; 					// Stan
	nBottleFeederTurnTableVelocityCV					:UDINT;						// Aktualna prędkość
	bBottleFeederTurnTableManualCmdStart				:BOOL; 					 	// Start 

	(***P01_PucksInserter***)
	// Podajnik opakowań
	iPucksInserterState									:INT;						// Stan
	sPucksInserterState									:STRING;					// Stan
	bPucksInserterRun									:BOOL;						// Cykl
	bPucksInserterHoming								:BOOL;						// Bazowanie 
	bPucksInserterHeightSet								:BOOL;						// Ustaw
	bPucksInserterIgnoreError							:BOOL;						// Ignoruj błędy
	bPucksInserterManualHammer							:BOOL;						// Wbijak	
	bPucksInserterManualTray							:BOOL;						// Tacka
	bPucksInserterManualGate1							:BOOL;						// Szlaban 1 - lewy
	bPucksInserterManualGate2							:BOOL;						// Szlaban 2 - prawy
	bPucksInserterManualFormGate						:BOOL;						// Szlaban formatki		
	bPucksInserterManualFormPositioning					:BOOL;						// Pozycjonowanie formatki	
	bPucksInserterManualWheelLeft						:BOOL;						// Karuzela - przód	
	bPucksInserterManualWheelRight						:BOOL;						// Karuzela - tył
	lrPucksInserterWheelPositionCV						:LREAl;						// Aktualna pozycja karuzeli


	//Transporter
	nPucksInserterConveyorVelocityCV					:UDINT;						// Aktualna prędkość
	bPucksInserterConveyorManualCmdStart				:BOOL; 					 	// Start 			
			
	// Wbijak na podnośniku
	lrPucksInserterHammerHeightCV						:LREAL;  					// Aktualna pozycja
    bPucksInserterManualHammerUp						:BOOL;  					// Do góry
    bPucksInserterManualHammerDown						:BOOL;  					// Na dół

	// Podajnik opakowań - stół							
	iPucksInserterTurnTableState						:INT; 					 	// Stan
	sPucksInserterTurnTableState						:STRING; 					// Stan
	nPucksInserterTurnTableVelocityCV					:UDINT;						// Aktualna prędkość
	bPucksInserterTurnTableManualCmdStart				:BOOL; 					 	// Start 
	
	
	//Stół popychający butelki Vasyl 27.05
	bPucksInserterPushTable_m1_ManualCmdStart				:BOOL; 					 	// Start silnik stołu pchającego - nr1
	bPucksInserterPushTable_m2_ManualCmdStart				:BOOL; 					 	// Start silnik stołu pchającego - nr2 
	bPucksInserterPushTable_m3_ManualCmdStart				:BOOL; 					 	// Start silnik stołu pchającego - nr3
	bPucksInserterPushTable_g1_ManualActuator				:BOOL;						// do usuniecia Siłownik stołu pchającego - nr1
	bPucksInserterPushTable_g2_ManualActuator				:BOOL;						// do usuniecia Siłownik stołu pchającego - nr2
	sPucksInserterPushTableState							:STRING;
	iPucksInserterPushTableState							:INT;
	sPucksInserterPushTableRollerState						:STRING;
	iPucksInserterPushTableRollerState						:INT;
	uiPucksInserterPushTable_m1_Velocity					:INT;
	uiPucksInserterPushTable_m2_Velocity					:INT;
	uiPucksInserterPushTable_m3_Velocity					:INT;
	
	(*****P01_Gates********)   
	// Szlaban przed dozownikami	
	iGateBeforeDispencersState							:INT; 						// Stan
	sGateBeforeDispencersState							:STRING; 					// Stan 
	bGateBeforeDispencersRun							:BOOL;						// Cykl
	bGateBeforeDispencersManualActuator					:BOOL;						// Manual - Szlaban
	
	(********P01_TwoPhasesBarriers*****)
	// Szlaban między dozownikami
	iBarrierBetweenDispencerState						:INT;						// Stan
	sBarrierBetweenDispencerState						:INT;						// Stan
	bBarrierBetweenDispencerRun							:BOOL;						// Cykl
	bBarrierBetweenDispencerManualActuator				:BOOL;						// Szlaban
	// Szlaban między wagami	
	iBarrierBetweenWeightState							:INT;						// Stan
	sBarrierBetweenWeightState							:INT;						// Stan
	bBarrierBetweenWeightRun							:BOOL;						// Cykl
	bBarrierBetweenWeightManualActuator					:BOOL;						// Szlaban
	// Szlaban przed wagą 1-4
	bGateBeforeWeight14Run								:BOOL;						// Cykl
	bGateBeforeWeight14ManualActuator					:BOOL;						// Szlaban
	// Szlaban przed wagą 5-6
	bGateBeforeWeight56Run								:BOOL;						// Cykl
	bGateBeforeWeight56ManualActuator					:BOOL;						// Szlaban
	// Szlaban przed podawaniem słoików	
	iBarrierLidFeederState								:INT;						// Stan
	sBarrierLidFeederState								:INT;						// Stan
	bBarrierLidFeederRun								:BOOL;						// Cykl
	bBarrierLidFeederManualActuator						:BOOL;						// Szlaban	
	// Szlaban przed podawaniem knotów	
	iBarrierWickFeederState								:INT;						// Stan
	sBarrierWickFeederState								:INT;						// Stan
	bBarrierWickFeederRun								:BOOL;						// Cykl
	bBarrierWickFeederManualActuator						:BOOL;						// Szlaban		
	//Szlaban pod robotem       	
	iGateRobotState										:INT; 						// Stan
	sGateRobotState										:STRING; 					// Stan
	bGateRobotEntranceRun								:BOOL;						// Cykl
	bGateRobotManualActuator							:BOOL;						// Szlaban
	
	(*[H]*P02_BottlePusher********)   
	// Wbijak butelek	
	iBottlePusherState									:INT; 						// [H] Stan
	sBottlePusherState									:STRING; 					// [H] Stan 
	bBottlePusherRun									:BOOL;						// [H] Cykl
	bBottlePusherManualActuator							:BOOL;						// [H] Manual - Szlaban	
	
	(*******P02_Dispencers******)
	// Przeciąganie formatek lewe
	iFormsDragingLeftState								:INT;						// Stan 
	sFormsDragingLeftState								:STRING;					// Stan  
	bFormsDragingLeftRun								:BOOL;						// Cykl
	bFormsDragingLeftHoming								:BOOL;						// Bazowanie 
	bFormsDragingLeftIgnoreError						:BOOL;						// Ignoruj błędy
	bFormsDragingLeftManualFork							:BOOL;						// Podnoszenie
	bFormsDragingLeftManualLeadBefore1					:BOOL;						// Prowadzenie 1
	bFormsDragingLeftManualLeadBefore2					:BOOL;						// Prowadzenie 2
	bFormsDragingLeftManualLeft							:BOOL;						// Przód
	bFormsDragingLeftManualRight						:BOOL;						// Tył
	lrFormsDragingLeftPositionCV						:LREAL;
	bFormsDispencersDragLeftMoveToEndPosition			:BOOL;
	// Przeciąganie formatek prawe	
	iFormsDragingRightState								:INT;						// Stan
	sFormsDragingRightState								:STRING;					// Stan 	
	bFormsDragingRightRun								:BOOL;						// Cykl
	bFormsDragingRightHoming							:BOOL;						// Bazowanie
	bFormsDragingRightIgnoreError						:BOOL;						// Ignoruj błędy
	bFormsDragingRightManualFork						:BOOL;						// Podnoszenie
	bFormsDragingRightManualLeadBefore1					:BOOL;						// Prowadzenie 1
	bFormsDragingRightManualLeadBefore2					:BOOL;						// Prowadzenie 2
	bFormsDragingRightManualLeft						:BOOL;						// Przód
	bFormsDragingRightManualRight						:BOOL;						// Tył
	lrFormsDragingRightPositionCV						:LREAL;
	bFormsDispencersDragRightMoveToEndPosition			:BOOL;
	//Dozowniki
 
	(**[L]**Synchronizacja dozowników**)
	//Przyśpieszenie obsługi dozowników
	//Synchronizacja potrzebna, po to aby wyświetlana aktualna pozycją się zgadzała
	//Po zaznaczeniu "synchronizacji jednego z dozowników" należy blokować przyciski aż zmienna "bDispencersSyncReady" będzie ustawiona (kilka sekund)
	//Na przykład: Jeżeli jest zaznaczone 1  i zostanie włączone "Dozuj" w PLC zostaje ustawiane "bDispencer1Dose"
	//Na przykład: Jeżeli jest zaznaczone SYNC 1 i 2 i zostanie włączone "Przeciągaj" w PLC zostaje ustawiane "bDispencer1PullingSlow","bDispencer2PullingSlow"
	//Na przykład: Jeżeli jest zaznaczone SYNC 3 i 4 i zostanie włączone "Dozuj" w PLC zostaje ustawiane "bDispencer3Dose","bDispencer4Dose"
	//itd. odpowiednio dla wszystkich przycisków trybu serwiswego
	bDispencer1Sync						: BOOL;			// Steruj 1 dozownikiem
	bDispencer2Sync						: BOOL;			// Steruj 2 dozownikiem
	bDispencer3Sync						: BOOL;			// Steruj 3 dozownikiem
	bDispencer4Sync						: BOOL;			// Steruj 4 dozownikiem
	bDispencer12Sync					: BOOL;			// Steruj 12 dozownikiem
	bDispencer34Sync					: BOOL;			// Steruj 34 dozownikiem
	bDispencer1234Sync					: BOOL;			// Steruj 1234 dozownikiem
	
	bDispencersSyncReady				: BOOL;			// Gotowość (odblokowane okienko sterowania)		

	// Zmienne ogólne okienka serwisowego, zależnie od zaznaczonych synchronizacji dozowników
    bDispencersDose                		: BOOL;   		// Dozuj
    bDispencersIgnoreErrors        		: BOOL;   		// Ignoruj błędy
    bDispencersHoming           		: BOOL;         // Bazowanie
    bDispencersManualDropCatcher 		: BOOL;         // Tacki
	bDispencersCleaning					: BOOL;			// Mycie
	lrDispencersManualOverride			: LREAL;		// [H] Prędkość
    bDispencersManualPistonBack     	: BOOL;   		// Tłok do góryw
    bDispencersManualPistonForward  	: BOOL;  		// Tłok w dół
    lrDispencersActPos             		: LREAL;  		// Aktualna pozycja tłoka
    bDispencersManualLifterUp       	: BOOL;   		// Podnośnik do góry
    bDispencersManualLifterDown   		: BOOL;   		// Podnośnik w dół
    lrDispencersLifterActPos      		: LREAL;  		// Aktualna pozycja 
    bDispencersPullingFast          	: BOOL;   		// Przeciąganie szybkie
    bDispencersPullingSlow         		: BOOL;   		// Przeciąganie wolne	
  	bDispencersPullingFastContinous		: BOOL;   		// Przeciąganie szybkie 30s
    bDispencersPullingSlowContinous		: BOOL;   		// Przeciąganie wolne 30s
    bDispencersManualSuckValve     		: BOOL;  	 	// Zawór ssący
    bDispencersManualDoseValve     		: BOOL;   		// Zawór tłoczący
	lrDispencersLifterSetPosStepMode	: LREAL;		// Skok ruchu [mm] (1.0-5.0)
	bDispencersLifterStepMode			: BOOL;			// Tryb krokowy
	//Ready position									
    bDispencersHeightSet          		: BOOL;   		// Ustaw
	(***Koniec synchronizacja dozowników**)	
	
	// [L] Mycie CIP 
	bDispencersCIP										: BOOL;						// [H] Włączone mycie CIP (stacje dozowników i chwytaków obniżają się)
	iDispencersCIP										: INT;						// [H] Zmienna pomocnicza od CIP (-1 pozycja dół, 0-Ruch, 1-pozycja górna)
	bDispencer12Cleaning								: BOOL;						// [H] Włączenie przeciągania dla dozownika 1 i 2 , wyłącza się po odciśnięciu przycisku
	bDispencer34Cleaning								: BOOL;						// [H] Włączenie przeciągania dla dozownika 3 i 4 , wyłącza się po odciśnięciu przycisku
	bDispencerManualDropCatcherSuck						: BOOL;						// Zasysanie z tacek

	//Podnośnik dozownika 1 2
    bDispencer12ManualLifterUp      					:BOOL;   					// Podnośnik 12 do góry
    bDispencer12ManualLifterDown  						:BOOL;   					// Podnośnik 12 w doł
	//Podnośnik dozownika 3 4
    bDispencer34ManualLifterUp      					:BOOL;   					// Podnośnik 34 do góry
    bDispencer34ManualLifterDown    					:BOOL;   					// Podnośnik 34 w dół

	lrDispencer12LifterActPos							:LREAL;						// Aktualna pozycja podnośnika dozownika 12
	lrDispencer12LifterSetPosStepMode					:LREAL;						// Krok przesuwania [mm] (1-5.0)
	bDispencer12LifterStepMode							:BOOL;						// Tryb krokowy
	
	lrDispencer34LifterActPos							:LREAL;						// Aktualna pozycja podnośnika dozownika 34
	lrDispencer34LifterSetPosStepMode					:LREAL;						// Krok przesuwania [mm] (1-5.0)
	bDispencer34LifterStepMode							:BOOL;						// Tryb krokowy

	
	bDispencer12LifterHeightSet							: BOOL;						// Ustaw podnośnik 12
	bDispencer34LifterHeightSet							: BOOL;						// Ustaw podnośnik 34
	
	//Dozownik 1                                        
	iDispencer1State									:INT; 						// Stan
	sDispencer1State									:STRING; 					// Stan
	bDispencer1IgnoreErrors								:BOOL; 						// Ignoruj błędy	
	bDispencer1Dose										:BOOL; 						// Dozuj 1
	lrDispencer1ActPos									:LREAL;						// Aktualna pozycja tłoka 1
	bDispencer1PullingFast								:BOOL;						// Przeciągnie szybkie 1
	bDispencer1PullingSlow								:BOOL;						// Przeciągnie wolne 1
	bDispencer1ManualPistonBack							:BOOL;						// Tłok 1 do góry
	bDispencer1ManualPistonForward						:BOOL;						// Tłok 1 w dół
	bDispencer1ManualSuckValve							:BOOL;						// Zawór ssący 1
	bDispencer1ManualDoseValve							:BOOL;						// Zawór dozujący 1

	//Dozownik 2                                        
	iDispencer2State									:INT; 						// Stan
	sDispencer2State									:STRING; 					// Stan
	bDispencer2IgnoreErrors								:BOOL; 						// Ignoruj błędy		
	bDispencer2Dose										:BOOL; 						// Dozuj 2
	lrDispencer2ActPos									:LREAL;						// Aktualna pozycja tłoka 2
	bDispencer2PullingFast								:BOOL;						// Przeciągnie szybkie 2
	bDispencer2PullingSlow								:BOOL;						// Przeciągnie wolne 2
	bDispencer2ManualPistonBack							:BOOL;						// Tłok 2 do góry
	bDispencer2ManualPistonForward						:BOOL;						// Tłok 2 w dół
	bDispencer2ManualSuckValve							:BOOL;						// Zawór ssący 2
	bDispencer2ManualDoseValve							:BOOL;						// Zawór dozujący 2

	//Dozownik 3                                        
	iDispencer3State									:INT; 						// Stan
	sDispencer3State									:STRING; 					// Stan
	bDispencer3IgnoreErrors								:BOOL; 						// Ignoruj błędy	
	bDispencer3Dose										:BOOL; 						// Dozuj 13
	lrDispencer3ActPos									:LREAL;						// Aktualna pozycja tłoka 3
	bDispencer3PullingFast								:BOOL;						// Przeciągnie szybkie 3
	bDispencer3PullingSlow								:BOOL;						// Przeciągnie wolne 3
	bDispencer3ManualPistonBack							:BOOL;						// Tłok 3 do góry
	bDispencer3ManualPistonForward						:BOOL;						// Tłok 3 w dół
	bDispencer3ManualSuckValve							:BOOL;						// Zawór ssący 3
	bDispencer3ManualDoseValve							:BOOL;						// Zawór dozujący 3
	                                                                                   
	//Dozownik 4                                        
	iDispencer4State									:INT; 						// Stan
	sDispencer4State									:STRING; 					// Stan
	bDispencer4IgnoreErrors								:BOOL; 						// Ignoruj błędy	
	bDispencer4Dose										:BOOL; 						// Dozuj 4
	lrDispencer4ActPos									:LREAL;						// Aktualna pozycja tłoka 4
	bDispencer4PullingFast								:BOOL;						// Przeciągnie szybkie 4
	bDispencer4PullingSlow								:BOOL;						// Przeciągnie wolne 4
	bDispencer4ManualPistonBack							:BOOL;						// Tłok 4 do góry
	bDispencer4ManualPistonForward						:BOOL;						// Tłok 4 w dół
	bDispencer4ManualSuckValve							:BOOL;						// Zawór ssący 4
	bDispencer4ManualDoseValve							:BOOL;						// Zawór dozujący 4
                                               
	//Podnośnik chwytaka                    	 
	lrDispencersCatchHeightCV							:LREAL;						// Aktualna wysokość chwytaka
    bDispencersCatchManualUp							:BOOL;  					// Do góry
    bDispencersCatchManualDown							:BOOL;  					// W dół
	bDispencersCatchHeightSet							:BOOL;						// Ustaw
	bDispencersCatchOpenCalibration						:BOOL;						// Kalibruj otwarcie
	bDispencersCatchCloseCalibration					:BOOL;						// Kalibruj zamknięcie
	
	//Podnośnik chwytaka i tacki 1                     	 
	iDispencersCatch1State								:INT;						// Stan
	sDispencersCatch1State								:STRING;					// Stan
	bDispencers1Catch									:BOOL;  					// Cykl
	bDispencersCatch1ManualActuator						:BOOL;  					// Chwytak
	
	//Podnośnik chwytaka i tacki 2                     	 
	iDispencersCatch2State								:INT;						// Stan
	sDispencersCatch2State								:STRING;					// Stan
	bDispencers2Catch									:BOOL;  					// Cykl
	bDispencersCatch2ManualActuator						:BOOL;  					// Chwytak
	
	//Podnośnik chwytaka i tacki 3                   	 
	bDispencers3Catch									:BOOL;  					// Stan
	iDispencersCatch3State								:INT;						// Stan
	sDispencersCatch3State								:STRING;					// Cykl
	bDispencersCatch3ManualActuator						:BOOL;  					// Chwytak

	//Podnośnik chwytaka i tacki 4                   	 
	iDispencersCatch4State								:INT;						// Stan
	sDispencersCatch4State								:STRING;					// Stan
	bDispencers4Catch									:BOOL;  					// Cykl
	bDispencersCatch4ManualActuator						:BOOL;  					// Chwytak

	//Zbiornik 1                                
	bTanksIgnoreError         					        :BOOL; 						// [H] Ignoruj błedy
    bTank1ManualMixer                 					:BOOL; 						// Mieszadło
    bTank1ManualHeater                					:BOOL; 						// Grzanie
    bTank1ManualSupplyPump            					:BOOL; 						// Pompa
    bTank1ManualPressure              					:BOOL; 						// Nadciśnienie
	lrTankHeatingTempCV									:LREAL;						// Temperatura zbiornika
	
	//Czujnik zbiornika 1
 	bTank1LevelSensorCalibrationLight					:BOOL;						// Kalibracja na pusto
	bTank1LevelSensorCalibrationDark					:BOOL;						// Kalibracja na pełno
	bHMITank1LevelSensorPumpOn							:BOOL;						// [I] Poziom (pompa załączona)
	iTank1LevelSensorValue								:INT; 						// Poziom [mm]
    bTank1LevelSensorHigh                               :BOOL;                      // [L] Zadany poziom ustawiony na 80%
    bTank1LevelSensorLow                                :BOOL;                      // [L] Zadany poziom ustawiony na 10%

	//Zbiornik 2  
    bTank2ManualMixer                 					:BOOL; 						// [H] Mieszadło
    bTank2ManualHeater                					:BOOL; 						// [H] Grzałka
    bTank2ManualSupplyPump            					:BOOL; 						// Pompa
    bTank2ManualPressure              					:BOOL; 						// [H] Nadciśnienie

	//Czujnik zbiornika 2
 	bTank2LevelSensorCalibrationLight					:BOOL;						// Kalibracja na pusto
	bTank2LevelSensorCalibrationDark					:BOOL;						// Kalibracja na pełno	
	bHMITank2LevelSensorPumpOn							:BOOL;						// [I] Poziom (pompa załączona)
	iTank2LevelSensorValue								:INT; 						// Poziom [mm]
     
	//Dodatkowe zbiorniki
	bHMITank3LevelSensorPumpOn							:BOOL;						// [I] Poziom (pompa załączona)
	iTank3LevelSensorValue								:INT; 						// Poziom [mm]
 	bHMITank4LevelSensorPumpOn							:BOOL;						// [I] Poziom (pompa załączona)
	iTank4LevelSensorValue								:INT; 						// Poziom [mm]
   
                                       	
	(*******P05_Weight*******)
	//Podnoszenie wag 
	iWeightLiftState									:INT;						// Stan 
	sWeightLiftState									:STRING;					// Stan 
	bWeightLiftRun										:BOOL;						// Cykl
	bWeightLiftHoming									:BOOL;						// Bazowanie
	//Waga 1 podnoszenie
	bWeight1ActuatorManualUp							: BOOL;						// Do góry
	bWeight1ActuatorManualDown							: BOOL;						// Na dół
	//Waga 2 podnoszenie
	bWeight2ActuatorManualUp							: BOOL;						// Do góry
	bWeight2ActuatorManualDown							: BOOL;						// Na dół
	//Waga 3 podnoszenie
	bWeight3ActuatorManualUp							: BOOL;						// Do góry
	bWeight3ActuatorManualDown							: BOOL;						// Na dół
	//Waga 4 podnoszenie	
	bWeight4ActuatorManualUp							: BOOL;						// Do góry
	bWeight4ActuatorManualDown							: BOOL;						// Na dół	
	//Waga 5 podnoszenie	
	bWeight5ActuatorManualUp							: BOOL;						// Do góry
	bWeight5ActuatorManualDown							: BOOL;						// Na dół	
	//Waga 6 podnoszenie	
	bWeight6ActuatorManualUp							: BOOL;						// Do góry
	bWeight6ActuatorManualDown							: BOOL;						// Na dół	
	
